# B&R Automation Studio project NAELD004C00R10L518F00 (part 13)

#### Act_OptP0932MagConv3FB.st
```iecst
ACTION Act_OptP0932MagConv3FB:

	//Magazine Conveyor
	IF tyP0932MagConv3.tyFB.tyBtnStop.bRtCompl = TRUE THEN
		eMagConv2Clp3Act	:= MagConv2ClpActStop;

		IF p_eMagConv2Clp3Stat = MagConv2ClpActStop AND p_eMagConv2Clp3Status = Done THEN
			eMagConv2Clp3Act	:= MagConv2ClpActIdle;

			tyP0932MagConv3.tyFB.tyBtnEnt.bRtCompl	:= FALSE;
			tyP0932MagConv3.tyFB.tyBtnEnt.bValue	:= FALSE;
			tyP0932MagConv3.tyFB.tyBtnEnt.bRtLk		:= FALSE;

			tyP0932MagConv3.tyFB.tyBtnExit.bRtCompl	:= FALSE;
			tyP0932MagConv3.tyFB.tyBtnExit.bValue	:= FALSE;
			tyP0932MagConv3.tyFB.tyBtnExit.bRtLk	:= FALSE;

			tyP0932MagConv3.tyFB.tyBtnStop.bRtCompl	:= FALSE;
			tyP0932MagConv3.tyFB.tyBtnStop.bValue	:= TRUE;
			tyP0932MagConv3.tyFB.tyBtnStop.bRtLk	:= TRUE;
		END_IF

	ELSIF tyP0932MagConv3.tyFB.tyBtnEnt.bRtCompl = TRUE THEN
		tyP0932MagConv3.tyFB.tyBtnEnt.bValue	:= TRUE;
		tyP0932MagConv3.tyFB.tyBtnEnt.bRtLk		:= TRUE;

		tyP0932MagConv3.tyFB.tyBtnStop.bValue	:= FALSE;
		tyP0932MagConv3.tyFB.tyBtnStop.bRtLk	:= FALSE;

		eMagConv2Clp3Act	:= MagConv2ClpActEnt;

		IF p_eMagConv2Clp3Stat = MagConv2ClpActEnt AND p_eMagConv2Clp3Status = Done THEN
			eMagConv2Clp3Act	:= MagConv2ClpActIdle;

			tyP0932MagConv3.tyFB.tyBtnEnt.bRtCompl	:= FALSE;

			tyP0932MagConv3.tyFB.tyBtnEnt.bValue	:= FALSE;
			tyP0932MagConv3.tyFB.tyBtnEnt.bRtLk		:= FALSE;

			tyP0932MagConv3.tyFB.tyBtnStop.bValue	:= TRUE;
			tyP0932MagConv3.tyFB.tyBtnStop.bRtLk	:= TRUE;
		END_IF

	ELSIF (p_eMagConv2Clp3Stat = MagConv2ClpActPreExit AND p_eMagConv2Clp3Status = Done) THEN
		eMagConv2Clp3Act	:= MagConv2ClpActIdle;

		tyP0932MagConv3.tyFB.tyBtnExit.bRtCompl	:= FALSE;

		tyP0932MagConv3.tyFB.tyBtnExit.bValue	:= FALSE;
		tyP0932MagConv3.tyFB.tyBtnExit.bRtLk	:= FALSE;

		tyP0932MagConv3.tyFB.tyBtnStop.bValue	:= TRUE;
		tyP0932MagConv3.tyFB.tyBtnStop.bRtLk	:= TRUE;

	ELSIF (p_eMagConv2Clp3Stat = MagConv2ClpActExit AND p_eMagConv2Clp3Status = Done) THEN
		eMagConv2Clp3Act	:= MagConv2ClpActIdle;

		tyP0932MagConv3.tyFB.tyBtnExit.bRtCompl	:= FALSE;

		tyP0932MagConv3.tyFB.tyBtnExit.bValue	:= FALSE;
		tyP0932MagConv3.tyFB.tyBtnExit.bRtLk	:= FALSE;

		tyP0932MagConv3.tyFB.tyBtnStop.bValue	:= TRUE;
		tyP0932MagConv3.tyFB.tyBtnStop.bRtLk	:= TRUE;

	ELSIF tyP0932MagConv3.tyFB.tyBtnExit.bRtCompl = TRUE THEN
		tyP0932MagConv3.tyFB.tyBtnExit.bRtCompl	:= FALSE;
		tyP0932MagConv3.tyFB.tyBtnExit.bValue	:= TRUE;
		tyP0932MagConv3.tyFB.tyBtnExit.bRtLk	:= TRUE;

		tyP0932MagConv3.tyFB.tyBtnStop.bValue	:= FALSE;
		tyP0932MagConv3.tyFB.tyBtnStop.bRtLk	:= FALSE;

		IF p_tyDI.bMagConvEntSen3  THEN
			eMagConv2Clp3Act	:= MagConv2ClpActExit;
		ELSE
			IF p_tyDI.bMagPresentSen3 THEN
				eMagConv2Clp3Act	:= MagConv2ClpActPreExit;
			ELSE
				eMagConv2Clp3Act	:= MagConv2ClpActExit;
			END_IF
		END_IF
	END_IF

	//Magazine Clamper
	IF tyP0932MagConv3.tyCom.tyBtnSwitch.bValue = FALSE THEN

		//Fixed/Bottom
		IF tyP0932MagConv3.tyFB.tyBtnFixedUnclamp.bRtCompl = TRUE THEN
			tyP0932MagConv3.tyFB.tyBtnFixedUnclamp.bRtCompl	:= FALSE;

			tyP0932MagConv3.tyFB.tyBtnFixedUnclamp.bValue	:= TRUE;
			tyP0932MagConv3.tyFB.tyBtnFixedClamp.bValue		:= FALSE;

		ELSIF tyP0932MagConv3.tyFB.tyBtnFixedClamp.bRtCompl = TRUE THEN
			tyP0932MagConv3.tyFB.tyBtnFixedClamp.bRtCompl	:= FALSE;

			tyP0932MagConv3.tyFB.tyBtnFixedClamp.bValue		:= TRUE;
			tyP0932MagConv3.tyFB.tyBtnFixedUnclamp.bValue	:= FALSE;

		END_IF

		//Remote/Top
		IF tyP0932MagConv3.tyFB.tyBtnRemoteUnclamp.bRtCompl = TRUE THEN
			tyP0932MagConv3.tyFB.tyBtnRemoteUnclamp.bRtCompl	:= FALSE;

			tyP0932MagConv3.tyFB.tyBtnRemoteUnclamp.bValue	:= TRUE;
			tyP0932MagConv3.tyFB.tyBtnRemoteClamp.bValue	:= FALSE;

		ELSIF tyP0932MagConv3.tyFB.tyBtnRemoteClamp.bRtCompl = TRUE THEN
			tyP0932MagConv3.tyFB.tyBtnRemoteClamp.bRtCompl	:= FALSE;

			tyP0932MagConv3.tyFB.tyBtnRemoteClamp.bValue	:= TRUE;
			tyP0932MagConv3.tyFB.tyBtnRemoteUnclamp.bValue	:= FALSE;

		END_IF

		//Selection
		IF tyP0932MagConv3.tyFB.tyBtnSelUnclamp.bRtCompl = TRUE THEN
			tyP0932MagConv3.tyFB.tyBtnSelUnclamp.bRtCompl	:= FALSE;

			tyP0932MagConv3.tyFB.tyBtnSelUnclamp.bValue	:= TRUE;
			tyP0932MagConv3.tyFB.tyBtnSelClamp.bValue	:= FALSE;

		ELSIF tyP0932MagConv3.tyFB.tyBtnSelClamp.bRtCompl = TRUE THEN
			tyP0932MagConv3.tyFB.tyBtnSelClamp.bRtCompl	:= FALSE;

			tyP0932MagConv3.tyFB.tyBtnSelClamp.bValue	:= TRUE;
			tyP0932MagConv3.tyFB.tyBtnSelUnclamp.bValue	:= FALSE;

		END_IF

		// Fixed Clamper
		IF tyP0932MagConv3.tyFB.tyBtnFixedUnclamp.bValue = TRUE THEN

			eMagConv2Clp3Act	:= MagConv2ClpActFixClprUnclamp;

			IF p_eMagConv2Clp3Stat = MagConv2ClpActFixClprUnclamp AND p_eMagConv2Clp3Status = Done THEN

				eMagConv2Clp3Act	:= MagConv2ClpActIdle;

				tyP0932MagConv3.tyFB.tyBtnFixedUnclamp.bValue	:= FALSE;

			ELSIF p_eMagConv2Clp3Status = Error THEN

				tyP0932MagConv3.tyFB.tyBtnFixedUnclamp.bValue	:= FALSE;

			END_IF

		ELSIF tyP0932MagConv3.tyFB.tyBtnFixedClamp.bValue = TRUE THEN
			eMagConv2Clp3Act	:= MagConv2ClpActFixClprClamp;

			IF p_eMagConv2Clp3Stat = MagConv2ClpActFixClprClamp AND p_eMagConv2Clp3Status = Done THEN

				eMagConv2Clp3Act	:= MagConv2ClpActIdle;

				tyP0932MagConv3.tyFB.tyBtnFixedClamp.bValue := FALSE;

			ELSIF p_eMagConv2Clp3Status = Error THEN

				tyP0932MagConv3.tyFB.tyBtnFixedClamp.bValue := FALSE;

			END_IF

		END_IF

		//Remote Clamper
		IF tyP0932MagConv3.tyFB.tyBtnRemoteUnclamp.bValue = TRUE THEN

			eMagConv2Clp3Act	:= MagConv2ClpActRmtClprUnclamp;

			IF p_eMagConv2Clp3Stat = MagConv2ClpActRmtClprUnclamp AND p_eMagConv2Clp3Status = Done THEN

				eMagConv2Clp3Act	:= MagConv2ClpActIdle;

				tyP0932MagConv3.tyFB.tyBtnRemoteUnclamp.bValue	:= FALSE;

			ELSIF p_eMagConv2Clp3Status = Error THEN

				tyP0932MagConv3.tyFB.tyBtnRemoteUnclamp.bValue	:= FALSE;

			END_IF

		ELSIF tyP0932MagConv3.tyFB.tyBtnRemoteClamp.bValue = TRUE THEN
			eMagConv2Clp3Act	:= MagConv2ClpActRmtClprClamp;

			IF p_eMagConv2Clp3Stat = MagConv2ClpActRmtClprClamp AND p_eMagConv2Clp3Status = Done THEN

				eMagConv2Clp3Act	:= MagConv2ClpActIdle;

				tyP0932MagConv3.tyFB.tyBtnRemoteClamp.bValue := FALSE;

			ELSIF p_eMagConv2Clp3Status = Error THEN
				tyP0932MagConv3.tyFB.tyBtnRemoteClamp.bValue := FALSE;

			END_IF

		END_IF

		//Selection Clamper
		IF tyP0932MagConv3.tyFB.tyBtnSelUnclamp.bValue = TRUE THEN

			eMagConvSelClp3Act	:= PneuActExt;

			IF p_eSelClamp3Stat = PneuActExt AND p_eSelClamp3Status = Done THEN

				eMagConvSelClp3Act	:= PneuActIdle;

				tyP0932MagConv3.tyFB.tyBtnSelUnclamp.bValue	:= FALSE;

			ELSIF p_eSelClamp3Status = Error THEN
				eMagConvSelClp3Act	:= PneuActIdle;
				tyP0932MagConv3.tyFB.tyBtnSelUnclamp.bValue	:= FALSE;

			END_IF

		ELSIF tyP0932MagConv3.tyFB.tyBtnSelClamp.bValue = TRUE THEN
			eMagConvSelClp3Act	:= PneuActRet;

			IF p_eSelClamp3Stat = PneuActRet AND p_eSelClamp3Status = Done THEN

				eMagConvSelClp3Act	:= PneuActIdle;

				tyP0932MagConv3.tyFB.tyBtnSelClamp.bValue	:= FALSE;

			ELSIF p_eSelClamp3Status = Error THEN
				eMagConvSelClp3Act	:= PneuActIdle;
				tyP0932MagConv3.tyFB.tyBtnSelClamp.bValue	:= FALSE;

			END_IF

		END_IF

		//Update Status
		tyP0932MagConv3.tyDC.tyBtnFixedUnclamp.bValue	:= NOT p_bMagConv2Clp3ClprFixClampCtrl;
		tyP0932MagConv3.tyDC.tyBtnFixedClamp.bValue		:= p_bMagConv2Clp3ClprFixClampCtrl;
		tyP0932MagConv3.tyDC.tyBtnRemoteUnclamp.bValue	:= NOT p_bMagConv2Clp3ClprRmtClampCtrl;
		tyP0932MagConv3.tyDC.tyBtnRemoteClamp.bValue	:= p_bMagConv2Clp3ClprRmtClampCtrl;

		tyP0932MagConv3.tyDC.tyBtnSelUnclamp.bRtCompl	:= FALSE;
		tyP0932MagConv3.tyDC.tyBtnSelClamp.bRtCompl		:= FALSE;
		tyP0932MagConv3.tyDC.tyBtnSelUnclamp.bValue	:= p_bSelClamp3RetCtrl;
		tyP0932MagConv3.tyDC.tyBtnSelClamp.bValue	:= p_bSelClamp3ExtCtrl;
	END_IF

	//Mask
	IF p_tyUsrMgmtCurrAccessRgt.bManualFBOnly THEN

		fUIInRtStatOff(ADR(tyP0932MagConv3.tyCom.tyBtnSwitch.uiMaskRtStat));

	ELSE

		IF p_eMagConv2Clp3Status = Error THEN

			fUIInRtStatOff(ADR(tyP0932MagConv3.tyFB.tyBtnEnt.uiMaskRtStat));
			fUIInRtStatOff(ADR(tyP0932MagConv3.tyFB.tyBtnExit.uiMaskRtStat));
			fUIInRtStatOff(ADR(tyP0932MagConv3.tyFB.tyBtnFixedClamp.uiMaskRtStat));
			fUIInRtStatOff(ADR(tyP0932MagConv3.tyFB.tyBtnFixedUnclamp.uiMaskRtStat));
			fUIInRtStatOff(ADR(tyP0932MagConv3.tyFB.tyBtnRemoteClamp.uiMaskRtStat));
			fUIInRtStatOff(ADR(tyP0932MagConv3.tyFB.tyBtnRemoteUnclamp.uiMaskRtStat));
			fUIInRtStatOff(ADR(tyP0932MagConv3.tyFB.tyBtnSelClamp.uiMaskRtStat));
			fUIInRtStatOff(ADR(tyP0932MagConv3.tyFB.tyBtnSelUnclamp.uiMaskRtStat));
			fUIInRtStatHide(ADR(tyP0932MagConv3.tyCom.tyBtnSwitch.uiMaskRtStat));

		ELSIF tyP0932MagConv3.tyFB.tyBtnEnt.bRtCompl = TRUE THEN

			fUIInRtStatHide(ADR(tyP0932MagConv3.tyFB.tyBtnEnt.uiMaskRtStat));
			fUIInRtStatOff(ADR(tyP0932MagConv3.tyFB.tyBtnExit.uiMaskRtStat));
			fUIInRtStatOff(ADR(tyP0932MagConv3.tyFB.tyBtnFixedClamp.uiMaskRtStat));
			fUIInRtStatOff(ADR(tyP0932MagConv3.tyFB.tyBtnFixedUnclamp.uiMaskRtStat));
			fUIInRtStatOff(ADR(tyP0932MagConv3.tyFB.tyBtnRemoteClamp.uiMaskRtStat));
			fUIInRtStatOff(ADR(tyP0932MagConv3.tyFB.tyBtnRemoteUnclamp.uiMaskRtStat));
			fUIInRtStatOff(ADR(tyP0932MagConv3.tyFB.tyBtnSelClamp.uiMaskRtStat));
			fUIInRtStatOff(ADR(tyP0932MagConv3.tyFB.tyBtnSelUnclamp.uiMaskRtStat));
			fUIInRtStatOff(ADR(tyP0932MagConv3.tyCom.tyBtnSwitch.uiMaskRtStat));

		ELSIF tyP0932MagConv3.tyFB.tyBtnExit.bRtCompl = TRUE THEN

			fUIInRtStatOff(ADR(tyP0932MagConv3.tyFB.tyBtnEnt.uiMaskRtStat));
			fUIInRtStatHide(ADR(tyP0932MagConv3.tyFB.tyBtnExit.uiMaskRtStat));
			fUIInRtStatOff(ADR(tyP0932MagConv3.tyFB.tyBtnFixedClamp.uiMaskRtStat));
			fUIInRtStatOff(ADR(tyP0932MagConv3.tyFB.tyBtnFixedUnclamp.uiMaskRtStat));
			fUIInRtStatOff(ADR(tyP0932MagConv3.tyFB.tyBtnRemoteClamp.uiMaskRtStat));
			fUIInRtStatOff(ADR(tyP0932MagConv3.tyFB.tyBtnRemoteUnclamp.uiMaskRtStat));
			fUIInRtStatOff(ADR(tyP0932MagConv3.tyFB.tyBtnSelClamp.uiMaskRtStat));
			fUIInRtStatOff(ADR(tyP0932MagConv3.tyFB.tyBtnSelUnclamp.uiMaskRtStat));
			fUIInRtStatOff(ADR(tyP0932MagConv3.tyCom.tyBtnSwitch.uiMaskRtStat));

		ELSIF tyP0932MagConv3.tyFB.tyBtnFixedClamp.bValue = TRUE OR tyP0932MagConv3.tyFB.tyBtnRemoteClamp.bValue = TRUE
			OR tyP0932MagConv3.tyFB.tyBtnFixedUnclamp.bValue = TRUE OR tyP0932MagConv3.tyFB.tyBtnRemoteUnclamp.bValue = TRUE
			OR tyP0932MagConv3.tyFB.tyBtnSelClamp.bValue = TRUE OR tyP0932MagConv3.tyFB.tyBtnSelUnclamp.bValue = TRUE
			THEN

			fUIInRtStatOff(ADR(tyP0932MagConv3.tyFB.tyBtnEnt.uiMaskRtStat));
			fUIInRtStatOff(ADR(tyP0932MagConv3.tyFB.tyBtnExit.uiMaskRtStat));
			fUIInRtStatHide(ADR(tyP0932MagConv3.tyFB.tyBtnFixedClamp.uiMaskRtStat));
			fUIInRtStatHide(ADR(tyP0932MagConv3.tyFB.tyBtnFixedUnclamp.uiMaskRtStat));
			fUIInRtStatHide(ADR(tyP0932MagConv3.tyFB.tyBtnRemoteClamp.uiMaskRtStat));
			fUIInRtStatHide(ADR(tyP0932MagConv3.tyFB.tyBtnRemoteUnclamp.uiMaskRtStat));
			fUIInRtStatHide(ADR(tyP0932MagConv3.tyFB.tyBtnSelClamp.uiMaskRtStat));
			fUIInRtStatHide(ADR(tyP0932MagConv3.tyFB.tyBtnSelUnclamp.uiMaskRtStat));
			fUIInRtStatOff(ADR(tyP0932MagConv3.tyCom.tyBtnSwitch.uiMaskRtStat));

		ELSE

			fUIInRtStatHide(ADR(tyP0932MagConv3.tyFB.tyBtnEnt.uiMaskRtStat));
			fUIInRtStatHide(ADR(tyP0932MagConv3.tyFB.tyBtnExit.uiMaskRtStat));
			fUIInRtStatHide(ADR(tyP0932MagConv3.tyFB.tyBtnFixedClamp.uiMaskRtStat));
			fUIInRtStatHide(ADR(tyP0932MagConv3.tyFB.tyBtnFixedUnclamp.uiMaskRtStat));
			fUIInRtStatHide(ADR(tyP0932MagConv3.tyFB.tyBtnRemoteClamp.uiMaskRtStat));
			fUIInRtStatHide(ADR(tyP0932MagConv3.tyFB.tyBtnRemoteUnclamp.uiMaskRtStat));
			fUIInRtStatHide(ADR(tyP0932MagConv3.tyFB.tyBtnSelClamp.uiMaskRtStat));
			fUIInRtStatHide(ADR(tyP0932MagConv3.tyFB.tyBtnSelUnclamp.uiMaskRtStat));
			fUIInRtStatHide(ADR(tyP0932MagConv3.tyCom.tyBtnSwitch.uiMaskRtStat));

		END_IF
	END_IF

	IF p_tyDI.bMagConvCAB717MagSen3 THEN
		fUIInRtStatOff(ADR(tyP0932MagConv3.tyFB.tyBtnSelClamp.uiMaskRtStat));
	END_IF

END_ACTION
```

#### Act_OptP0932MagConv3FBStat.st
```iecst
ACTION Act_OptP0932MagConv3FBStat:

	IF tyP0932MagConv3.tyFB.tyBtnFixedClamp.bValue = TRUE OR tyP0932MagConv3.tyFB.tyBtnRemoteClamp.bValue = TRUE
		OR tyP0932MagConv3.tyFB.tyBtnFixedUnclamp.bValue = TRUE OR tyP0932MagConv3.tyFB.tyBtnRemoteUnclamp.bValue = TRUE
		THEN
		tyP0932MagConv3.tyFB.tyStringStat.sValue	:= p_sMagConv2Clp3StatTxt;
	ELSIF tyP0932MagConv3.tyFB.tyBtnSelUnclamp.bValue = TRUE OR tyP0932MagConv3.tyFB.tyBtnSelClamp.bValue = TRUE
		THEN
		tyP0932MagConv3.tyFB.tyStringStat.sValue	:= p_sSelClamp3StatTxt;
	END_IF
END_ACTION
```

#### Act_OptP0932MagConv3Sen.st
```iecst
ACTION Act_OptP0932MagConv3Sen:

	tyP0932MagConv3.tyCom.tyBtnMagPresentSen.bValue			:= p_tyDI.bMagPresentSen3;
	tyP0932MagConv3.tyCom.tyBtnMagConvEntSen.bValue			:= p_tyDI.bMagConvEntSen3;
	tyP0932MagConv3.tyCom.tyBtnMagAIVPosSen1.bValue			:= p_tyDI.bMag3AGVInPosSen1;
	tyP0932MagConv3.tyCom.tyBtnMagAIVPosSen2.bValue			:= p_tyDI.bMag3AGVInPosSen2;
	tyP0932MagConv3.tyCom.tyBtnMagOrientationChkSen1.bValue	:= p_tyDI.bMag3OrientChkSen1;
	tyP0932MagConv3.tyCom.tyBtnMagOrientationChkSen2.bValue	:= p_tyDI.bMag3OrientChkSen2;

	tyP0932MagConv3.tyCom.tyBtnFixedClampRS.bValue			:= p_tyDI.bMag3FixedClampRS;
	tyP0932MagConv3.tyCom.tyBtnFixedUnclampRS.bValue		:= p_tyDI.bMag3FixedUnclampRS;
	tyP0932MagConv3.tyCom.tyBtnRemoteClampRS.bValue			:= p_tyDI.bMag3RemoteClampRS;
	tyP0932MagConv3.tyCom.tyBtnRemoteUnclampRS.bValue		:= p_tyDI.bMag3RemoteUnclampRS;

	tyP0932MagConv3.tyCom.tyBtnSelUnclampRS.bValue			:= p_tyDI.bMag3SelUnClampRS;

	tyP0932MagConv3.tyCom.tyBtnCAB717Sen.bValue				:= p_tyDI.bMagConvCAB717MagSen3;
	tyP0932MagConv3.tyCom.tyBtnHeightSen.bValue				:= p_tyDI.bMagConvHeightSen3 OR p_tyDI.bHighMagDetSen3;
	tyP0932MagConv3.tyCom.tyBtnMagSmallSen.bValue			:= p_tyDI.bMagConvSmallMagSen3;
	tyP0932MagConv3.tyCom.tyBtnMagLargeSen.bValue			:= p_tyDI.bMagConvLargeMagSen3;
	tyP0932MagConv3.tyCom.tyBtnMagDetSen.bValue				:= p_tyDI.bMag3FixedSideDetect;

	//Machine Bitmap //23
//	IF p_tyNtParamCurr.bMagAutoVerifyPrep = FALSE THEN
//		IF tyP0932MagConv3.tyFB.tyBtnFixedClamp.bRtCompl OR  tyP0932MagConv3.tyFB.tyBtnRemoteClamp.bRtCompl
//			OR tyP0932MagConv3.tyDC.tyBtnFixedClamp.bRtCompl OR tyP0932MagConv3.tyDC.tyBtnRemoteClamp.bRtCompl  THEN
//
//			tyP0932MagConv3.tyCom.tyBitmapMc.uiValueIdx	:= 2;
//
//		ELSIF tyP0932MagConv3.tyFB.tyBtnFixedUnclamp.bRtCompl OR tyP0932MagConv3.tyFB.tyBtnRemoteUnclamp.bRtCompl
//			OR tyP0932MagConv3.tyDC.tyBtnFixedUnclamp.bRtCompl OR tyP0932MagConv3.tyDC.tyBtnRemoteUnclamp.bRtCompl  THEN
//
//			tyP0932MagConv3.tyCom.tyBitmapMc.uiValueIdx	:= 1;
//
//		ELSIF tyP0932MagConv3.tyFB.tyBtnEnt.bRtCompl OR tyP0932MagConv3.tyFB.tyBtnExit.bRtCompl OR tyP0932MagConv3.tyFB.tyBtnStop.bRtCompl
//			OR tyP0932MagConv3.tyDC.tyBtnMagIn.bRtCompl OR tyP0932MagConv3.tyDC.tyBtnMagOut.bRtCompl OR tyP0932MagConv3.tyDC.tyBtnStop.bRtCompl THEN
//
//			tyP0932MagConv3.tyCom.tyBitmapMc.uiValueIdx	:= 0;
//
//		END_IF

	IF p_tyNtParamCurr.eProjMag = LDMagTriple AND p_tyNtParamCurr.bProjCurtainSenPrep = FALSE AND p_tyNtParamCurr.eCustomerReq <> Siemens AND p_tyNtParamCurr.eCustomerReq <> We_Fabricate  THEN
		IF tyP0932MagConv3.tyFB.tyBtnFixedClamp.bRtCompl
			OR tyP0932MagConv3.tyDC.tyBtnFixedClamp.bRtCompl THEN

			tyP0932MagConv3.tyCom.tyBitmapMc.uiValueIdx	:= 2;

		ELSIF tyP0932MagConv3.tyFB.tyBtnFixedUnclamp.bRtCompl
			OR tyP0932MagConv3.tyDC.tyBtnFixedUnclamp.bRtCompl THEN

			tyP0932MagConv3.tyCom.tyBitmapMc.uiValueIdx	:= 1;

		ELSIF tyP0932MagConv3.tyFB.tyBtnRemoteClamp.bRtCompl
			OR tyP0932MagConv3.tyDC.tyBtnRemoteClamp.bRtCompl THEN

			tyP0932MagConv3.tyCom.tyBitmapMc.uiValueIdx	:= 14;

		ELSIF tyP0932MagConv3.tyFB.tyBtnRemoteUnclamp.bRtCompl
			OR tyP0932MagConv3.tyDC.tyBtnRemoteUnclamp.bRtCompl THEN

			tyP0932MagConv3.tyCom.tyBitmapMc.uiValueIdx	:= 13;

		ELSIF tyP0932MagConv3.tyFB.tyBtnSelClamp.bRtCompl
			OR tyP0932MagConv3.tyDC.tyBtnSelClamp.bRtCompl THEN

			tyP0932MagConv3.tyCom.tyBitmapMc.uiValueIdx	:= 20;

		ELSIF tyP0932MagConv3.tyFB.tyBtnSelUnclamp.bRtCompl
			OR tyP0932MagConv3.tyDC.tyBtnSelUnclamp.bRtCompl THEN

			tyP0932MagConv3.tyCom.tyBitmapMc.uiValueIdx	:= 19;

		ELSIF tyP0932MagConv3.tyFB.tyBtnEnt.bRtCompl OR tyP0932MagConv3.tyFB.tyBtnExit.bRtCompl OR tyP0932MagConv3.tyFB.tyBtnStop.bRtCompl
			OR tyP0932MagConv3.tyDC.tyBtnMagIn.bRtCompl OR tyP0932MagConv3.tyDC.tyBtnMagOut.bRtCompl OR tyP0932MagConv3.tyDC.tyBtnStop.bRtCompl THEN

			tyP0932MagConv3.tyCom.tyBitmapMc.uiValueIdx	:= 0;

		END_IF
	ELSIF p_tyNtParamCurr.eProjMag = LDMagTriple AND p_tyNtParamCurr.bProjCurtainSenPrep OR p_tyNtParamCurr.eCustomerReq = Siemens OR p_tyNtParamCurr.eCustomerReq = We_Fabricate THEN
		tyP0932MagConv3.tyCom.tyBitmapMc.uiValueIdx	:= 386-23;

	ELSIF p_tyNtParamCurr.eProjMag = LDMagQuadruple AND p_tyNtParamCurr.bMagAutoVerifyPrep THEN
		IF tyP0932MagConv3.tyFB.tyBtnFixedClamp.bRtCompl
			OR tyP0932MagConv3.tyDC.tyBtnFixedClamp.bRtCompl THEN

			tyP0932MagConv3.tyCom.tyBitmapMc.uiValueIdx	:= 111;

		ELSIF tyP0932MagConv3.tyFB.tyBtnFixedUnclamp.bRtCompl
			OR tyP0932MagConv3.tyDC.tyBtnFixedUnclamp.bRtCompl THEN

			tyP0932MagConv3.tyCom.tyBitmapMc.uiValueIdx	:= 110;

		ELSIF tyP0932MagConv3.tyFB.tyBtnRemoteClamp.bRtCompl
			OR tyP0932MagConv3.tyDC.tyBtnRemoteClamp.bRtCompl THEN

			tyP0932MagConv3.tyCom.tyBitmapMc.uiValueIdx	:= 113;

		ELSIF tyP0932MagConv3.tyFB.tyBtnRemoteUnclamp.bRtCompl
			OR tyP0932MagConv3.tyDC.tyBtnRemoteUnclamp.bRtCompl THEN

			tyP0932MagConv3.tyCom.tyBitmapMc.uiValueIdx	:= 112;

		ELSIF tyP0932MagConv3.tyFB.tyBtnSelClamp.bRtCompl
			OR tyP0932MagConv3.tyDC.tyBtnSelClamp.bRtCompl THEN

			tyP0932MagConv3.tyCom.tyBitmapMc.uiValueIdx	:= 115;

		ELSIF tyP0932MagConv3.tyFB.tyBtnSelUnclamp.bRtCompl
			OR tyP0932MagConv3.tyDC.tyBtnSelUnclamp.bRtCompl THEN

			tyP0932MagConv3.tyCom.tyBitmapMc.uiValueIdx	:= 114;

		ELSIF tyP0932MagConv3.tyFB.tyBtnEnt.bRtCompl OR tyP0932MagConv3.tyFB.tyBtnExit.bRtCompl OR tyP0932MagConv3.tyFB.tyBtnStop.bRtCompl
			OR tyP0932MagConv3.tyDC.tyBtnMagIn.bRtCompl OR tyP0932MagConv3.tyDC.tyBtnMagOut.bRtCompl OR tyP0932MagConv3.tyDC.tyBtnStop.bRtCompl THEN

			tyP0932MagConv3.tyCom.tyBitmapMc.uiValueIdx	:= 109;

		END_IF
	END_IF

	IF p_tyNtParamCurr.eProjMag = LDMagTriple AND p_tyNtParamCurr.bMagAutoVerifyPrep = FALSE AND p_tyNtParamCurr.bProjMotorizedPullerPrep = FALSE THEN
		IF tyP0932MagConv3.tyCom.tyBitmapMc.uiValueIdx < 100 THEN
			tyP0932MagConv3.tyCom.tyBitmapMc.uiValueIdx	:= tyP0932MagConv3.tyCom.tyBitmapMc.uiValueIdx + 100;
		END_IF
	ELSIF p_tyNtParamCurr.eProjMag = LDMagDual AND p_tyNtParamCurr.bMagAutoVerifyPrep = TRUE THEN
		IF tyP0932MagConv3.tyCom.tyBitmapMc.uiValueIdx < 200 THEN
			tyP0932MagConv3.tyCom.tyBitmapMc.uiValueIdx	:= tyP0932MagConv3.tyCom.tyBitmapMc.uiValueIdx + 200;
		END_IF
	ELSIF p_tyNtParamCurr.eProjMag = LDMagTriple AND p_tyNtParamCurr.bMagAutoVerifyPrep = FALSE AND p_tyNtParamCurr.bProjMotorizedPullerPrep = TRUE THEN
			IF tyP0932MagConv3.tyCom.tyBitmapMc.uiValueIdx < 300 THEN
				tyP0932MagConv3.tyCom.tyBitmapMc.uiValueIdx	:= tyP0932MagConv3.tyCom.tyBitmapMc.uiValueIdx + 300;
			END_IF
	END_IF

END_ACTION
```

#### Act_OptP0932Navi.st
```iecst
ACTION Act_OptP0932Navi:

	CASE p_tyNtParamCurr.eProjMag OF
		LDMagDual:
			IF tyP0932MagConv3.tyNavi3Lyr3.tyBtnBack.bRtCompl = TRUE THEN
				tyP0932MagConv3.tyNavi3Lyr3.tyBtnBack.bRtCompl	:= FALSE;
				tyP0932MagConv3.tyNavi3Lyr3.tyBtnBack.bValue	:= FALSE;

				eChgPage	:= UIP0920MtrNPneuCtrl;

				bDispMagConv1	:= FALSE;
				bDispMagConv2	:= FALSE;
				bDispMagConv3	:= TRUE;
				bDispMagConv4	:= FALSE;

			ELSIF tyP0932MagConv3.tyNavi3Lyr3.tyBtnLeft.bRtCompl = TRUE
				OR tyP0932MagConv3.tyNavi3Lyr3.tyBtnRgt.bRtCompl = TRUE
				THEN
				tyP0932MagConv3.tyNavi3Lyr3.tyBtnLeft.bRtCompl			:= FALSE;
				tyP0932MagConv3.tyNavi3Lyr3.tyBtnLeft.bValue			:= FALSE;
				tyP0932MagConv3.tyNavi3Lyr3.tyBtnRgt.bRtCompl			:= FALSE;
				tyP0932MagConv3.tyNavi3Lyr3.tyBtnRgt.bValue				:= FALSE;
				eChgPage												:= UIP0931MagConv2;
				bDispMagConv1	:= FALSE;
				bDispMagConv2	:= TRUE;
				bDispMagConv3	:= FALSE;
				bDispMagConv4	:= FALSE;
			END_IF

		LDMagTriple:
			IF tyP0932MagConv3.tyNavi3Lyr3.tyBtnBack.bRtCompl = TRUE THEN
				tyP0932MagConv3.tyNavi3Lyr3.tyBtnBack.bRtCompl	:= FALSE;
				tyP0932MagConv3.tyNavi3Lyr3.tyBtnBack.bValue	:= FALSE;

				eChgPage	:= UIP0920MtrNPneuCtrl;

				bDispMagConv1	:= FALSE;
				bDispMagConv2	:= FALSE;
				bDispMagConv3	:= TRUE;
				bDispMagConv4	:= FALSE;

			ELSIF tyP0932MagConv3.tyNavi3Lyr3.tyBtnLeft.bRtCompl = TRUE THEN
				tyP0932MagConv3.tyNavi3Lyr3.tyBtnLeft.bRtCompl			:= FALSE;
				tyP0932MagConv3.tyNavi3Lyr3.tyBtnLeft.bValue			:= FALSE;
				eChgPage												:= UIP0931MagConv2;
				bDispMagConv1	:= FALSE;
				bDispMagConv2	:= TRUE;
				bDispMagConv3	:= FALSE;
				bDispMagConv4	:= FALSE;

			ELSIF tyP0932MagConv3.tyNavi3Lyr3.tyBtnRgt.bRtCompl = TRUE THEN
				tyP0932MagConv3.tyNavi3Lyr3.tyBtnRgt.bRtCompl			:= FALSE;
				tyP0932MagConv3.tyNavi3Lyr3.tyBtnRgt.bValue				:= FALSE;
				eChgPage												:= UIP0930MagConv1;
				bDispMagConv1	:= TRUE;
				bDispMagConv2	:= FALSE;
				bDispMagConv3	:= FALSE;
				bDispMagConv4	:= FALSE;
			END_IF

		LDMagQuadruple:
			IF tyP0932MagConv3.tyNavi4Lyr3.tyBtnBack.bRtCompl = TRUE THEN
				tyP0932MagConv3.tyNavi4Lyr3.tyBtnBack.bRtCompl	:= FALSE;
				tyP0932MagConv3.tyNavi4Lyr3.tyBtnBack.bValue	:= FALSE;

				eChgPage	:= UIP0920MtrNPneuCtrl;
				bDispMagConv1	:= FALSE;
				bDispMagConv2	:= FALSE;
				bDispMagConv3	:= TRUE;
				bDispMagConv4	:= FALSE;

			ELSIF tyP0932MagConv3.tyNavi4Lyr3.tyBtnLeft.bRtCompl = TRUE THEN
				tyP0932MagConv3.tyNavi4Lyr3.tyBtnLeft.bRtCompl			:= FALSE;
				tyP0932MagConv3.tyNavi4Lyr3.tyBtnLeft.bValue			:= FALSE;
				eChgPage												:= UIP0931MagConv2;
				bDispMagConv1	:= FALSE;
				bDispMagConv2	:= TRUE;
				bDispMagConv3	:= FALSE;
				bDispMagConv4	:= FALSE;

			ELSIF tyP0932MagConv3.tyNavi4Lyr3.tyBtnRgt.bRtCompl = TRUE THEN
				tyP0932MagConv3.tyNavi4Lyr3.tyBtnRgt.bRtCompl			:= FALSE;
				tyP0932MagConv3.tyNavi4Lyr3.tyBtnRgt.bValue				:= FALSE;
				eChgPage												:= UIP0939MagConv4;
				bDispMagConv1	:= FALSE;
				bDispMagConv2	:= FALSE;
				bDispMagConv3	:= FALSE;
				bDispMagConv4	:= TRUE;
			END_IF
	END_CASE

END_ACTION
```

#### Act_OptP0932RstMnl.st
```iecst
ACTION Act_OptP0932RstMnl:

	IF EDGEPOS((bManualMod = FALSE) OR (p_eMagConv2Clp3Status = Error)) THEN

		eMagConv2Clp3Act	:= MagConv2ClpActIdle;
		eMagConvSelClp3Act	:= PneuActIdle;
		//Magazine Conveyor
		//FB
		tyP0932MagConv3.tyFB.tyBtnEnt.bRtCompl				:= FALSE;
		tyP0932MagConv3.tyFB.tyBtnExit.bRtCompl				:= FALSE;
		tyP0932MagConv3.tyFB.tyBtnStop.bRtCompl				:= FALSE;

		tyP0932MagConv3.tyFB.tyBtnEnt.bValue				:= FALSE;
		tyP0932MagConv3.tyFB.tyBtnExit.bValue				:= FALSE;
		tyP0932MagConv3.tyFB.tyBtnStop.bValue				:= TRUE;

		tyP0932MagConv3.tyFB.tyBtnEnt.bRtLk					:= FALSE;
		tyP0932MagConv3.tyFB.tyBtnExit.bRtLk				:= FALSE;
		tyP0932MagConv3.tyFB.tyBtnStop.bRtLk				:= TRUE;

		tyP0932MagConv3.tyFB.tyBtnEnt.uiMaskRtStat.0		:= TRUE;
		tyP0932MagConv3.tyFB.tyBtnExit.uiMaskRtStat.0		:= TRUE;
		tyP0932MagConv3.tyCom.tyBtnSwitch.uiMaskRtStat.0	:= TRUE;

		//Direct
		tyP0932MagConv3.tyDC.tyBtnMagIn.bRtCompl			:= FALSE;
		tyP0932MagConv3.tyDC.tyBtnMagOut.bRtCompl			:= FALSE;
		tyP0932MagConv3.tyDC.tyBtnStop.bRtCompl				:= FALSE;

		tyP0932MagConv3.tyDC.tyBtnMagIn.bValue				:= FALSE;
		tyP0932MagConv3.tyDC.tyBtnMagOut.bValue				:= FALSE;
		tyP0932MagConv3.tyDC.tyBtnStop.bValue				:= TRUE;

		tyP0932MagConv3.tyDC.tyBtnMagIn.bRtLk				:= FALSE;
		tyP0932MagConv3.tyDC.tyBtnMagOut.bRtLk				:= FALSE;
		tyP0932MagConv3.tyDC.tyBtnStop.bRtLk				:= TRUE;

		tyP0932MagConv3.tyDC.tyBtnMagIn.uiMaskRtStat.0		:= TRUE;
		tyP0932MagConv3.tyDC.tyBtnMagOut.uiMaskRtStat.0		:= TRUE;
		tyP0932MagConv3.tyCom.tyBtnSwitch.uiMaskRtStat.0	:= TRUE;

		//Magazine Clamper
		//FB
		//Fixed/Bottom
		tyP0932MagConv3.tyFB.tyBtnFixedClamp.bRtCompl			:= FALSE;
		tyP0932MagConv3.tyFB.tyBtnFixedUnclamp.bRtCompl			:= FALSE;

		tyP0932MagConv3.tyFB.tyBtnFixedClamp.bValue				:= FALSE;
		tyP0932MagConv3.tyFB.tyBtnFixedUnclamp.bValue			:= FALSE;

		//Remote/Top
		tyP0932MagConv3.tyFB.tyBtnRemoteClamp.bRtCompl			:= FALSE;
		tyP0932MagConv3.tyFB.tyBtnRemoteUnclamp.bRtCompl		:= FALSE;

		tyP0932MagConv3.tyFB.tyBtnRemoteClamp.bValue			:= FALSE;
		tyP0932MagConv3.tyFB.tyBtnRemoteUnclamp.bValue			:= FALSE;

		//Selection
		tyP0932MagConv3.tyFB.tyBtnSelClamp.bRtCompl			:= FALSE;
		tyP0932MagConv3.tyFB.tyBtnSelUnclamp.bRtCompl		:= FALSE;

		tyP0932MagConv3.tyFB.tyBtnSelClamp.bValue			:= FALSE;
		tyP0932MagConv3.tyFB.tyBtnSelUnclamp.bValue			:= FALSE;

		tyP0932MagConv3.tyFB.tyBtnFixedClamp.uiMaskRtStat.0		:= TRUE;
		tyP0932MagConv3.tyFB.tyBtnFixedUnclamp.uiMaskRtStat.0	:= TRUE;
		tyP0932MagConv3.tyFB.tyBtnRemoteClamp.uiMaskRtStat.0	:= TRUE;
		tyP0932MagConv3.tyFB.tyBtnRemoteUnclamp.uiMaskRtStat.0	:= TRUE;
		tyP0932MagConv3.tyFB.tyBtnSelClamp.uiMaskRtStat.0		:= TRUE;
		tyP0932MagConv3.tyFB.tyBtnSelUnclamp.uiMaskRtStat.0		:= TRUE;

		tyP0932MagConv3.tyCom.tyBtnSwitch.uiMaskRtStat.0		:= TRUE;

		//Direct
		//Fixed/Bottom
		tyP0932MagConv3.tyDC.tyBtnFixedClamp.bRtCompl			:= FALSE;
		tyP0932MagConv3.tyDC.tyBtnFixedUnclamp.bRtCompl			:= FALSE;

		tyP0932MagConv3.tyDC.tyBtnFixedClamp.bValue				:= FALSE;
		tyP0932MagConv3.tyDC.tyBtnFixedUnclamp.bValue			:= FALSE;

		//Remote/Top
		tyP0932MagConv3.tyDC.tyBtnRemoteClamp.bRtCompl			:= FALSE;
		tyP0932MagConv3.tyDC.tyBtnRemoteUnclamp.bRtCompl		:= FALSE;

		tyP0932MagConv3.tyDC.tyBtnRemoteClamp.bValue			:= FALSE;
		tyP0932MagConv3.tyDC.tyBtnRemoteUnclamp.bValue			:= FALSE;

		//Selection
		tyP0932MagConv3.tyDC.tyBtnSelClamp.bRtCompl				:= FALSE;
		tyP0932MagConv3.tyDC.tyBtnSelUnclamp.bRtCompl			:= FALSE;

		tyP0932MagConv3.tyDC.tyBtnSelClamp.bValue				:= FALSE;
		tyP0932MagConv3.tyDC.tyBtnSelUnclamp.bValue				:= FALSE;

		tyP0932MagConv3.tyDC.tyBtnFixedClamp.uiMaskRtStat.0		:= TRUE;
		tyP0932MagConv3.tyDC.tyBtnFixedUnclamp.uiMaskRtStat.0	:= TRUE;
		tyP0932MagConv3.tyDC.tyBtnRemoteClamp.uiMaskRtStat.0	:= TRUE;
		tyP0932MagConv3.tyDC.tyBtnRemoteUnclamp.uiMaskRtStat.0	:= TRUE;
		tyP0932MagConv3.tyDC.tyBtnSelClamp.uiMaskRtStat.0		:= TRUE;
		tyP0932MagConv3.tyDC.tyBtnSelUnclamp.uiMaskRtStat.0		:= TRUE;

		tyP0932MagConv3.tyCom.tyBtnSwitch.uiMaskRtStat.0		:= TRUE;

	END_IF

	IF EDGEPOS(bManualMod = FALSE) THEN
		tyP0932MagConv3.tyCom.tyBtnSwitch.bValue := FALSE;

		IF p_tyNtParamCurr.bMagAutoVerifyPrep = FALSE THEN
			fUIInRtStatHide(ADR(tyP0932MagConv3.tyDC.tyLyrWithoutSelClamp.uiRtStat));
			fUIInRtStatOff(ADR(tyP0932MagConv3.tyFB.tyLyrWithoutSelClamp.uiRtStat));
		ELSE

			fUIInRtStatHide(ADR(tyP0932MagConv3.tyDC.tyLyr.uiRtStat));
			fUIInRtStatOff(ADR(tyP0932MagConv3.tyFB.tyLyr.uiRtStat));
		END_IF

	END_IF

END_ACTION
```

#### Act_EntP0933Disp.st
```iecst
ACTION Act_EntP0933Disp:

	//Access Address
	p_tyC0002FullMask ACCESS ADR(tyP0933PullConv.tyFullMaskHide);

	p_tyC0004Navi ACCESS ADR(tyP0933PullConv.tyNaviBack);

	p_tyC0005Main ACCESS ADR(tyCommon.tyMain);

	p_tyC0007Notif ACCESS ADR(tyCommon.tyNotif);

	p_tyC0008MsgBox ACCESS ADR(tyP0933PullConv.tyMsgBoxHide);

	p_tyC0009Info ACCESS ADR(tyCommon.tyInfo);

	p_tyP0933PullConvCom ACCESS ADR(tyP0933PullConv.tyCom);
	p_tyP0933PullConvDC ACCESS ADR(tyP0933PullConv.tyDC);
	p_tyP0933PullConvFB ACCESS ADR(tyP0933PullConv.tyFB);

	//Display
	IF p_tyProdRcpCurrRcp0.diMtrPshrExtSpd <> 0 THEN
		tyP0933PullConv.tyFB.tyNumExtSpd.diValue			:= p_tyProdRcpCurrRcp0.diMtrPshrExtSpd;
	ELSE
		tyP0933PullConv.tyFB.tyNumExtSpd.diValue			:= p_tyNtParamCurr.tyProdRcpMtrPshrExtSpd.diMax/2;
	END_IF

	IF p_tyProdRcpCurrRcp0.diMtrPshrExtTorq <> 0 THEN
		tyP0933PullConv.tyFB.tyNumExtTorqPercent.diValue	:= p_tyProdRcpCurrRcp0.diMtrPshrExtTorq;
	ELSE
		tyP0933PullConv.tyFB.tyNumExtTorqPercent.diValue	:= p_tyNtParamCurr.tyProdRcpMtrPshrExtTorq.diMax/2;
	END_IF
END_ACTION
```

#### Act_OptP0933Navi.st
```iecst
ACTION Act_OptP0933Navi:

	IF tyP0933PullConv.tyNaviBack.tyBtnBack.bRtCompl = TRUE THEN
		tyP0933PullConv.tyNaviBack.tyBtnBack.bRtCompl	:= FALSE;
		tyP0933PullConv.tyNaviBack.tyBtnBack.bValue		:= FALSE;

		eChgPage	:= UIP0920MtrNPneuCtrl;
	END_IF

END_ACTION
```

#### Act_OptP0933FullMask.st
```iecst
ACTION Act_OptP0933FullMask:

	IF eCurrPage = UIP0933PullConv THEN

		IF p_tyDI.bEStopSig = FALSE THEN
			p_tyC0002FullMask ACCESS ADR(tyP0933PullConv.tyFullMaskEStop);

		ELSIF p_tyDI.bCoverSWSig = FALSE THEN
			p_tyC0002FullMask ACCESS ADR(tyP0933PullConv.tyFullMaskCWSig);

		ELSIF p_tyDI.bSafetyRlySig = FALSE THEN
			p_tyC0002FullMask ACCESS ADR(tyP0933PullConv.tyFullMaskSafetyRly);

		ELSIF p_tyNtParamCurr.bAWPrep AND  p_tyNtParamCurr.bAWPusherPrep
			AND p_tyMcParamCurr.bAWDis = FALSE
			AND p_bAWOpenIsHomed = FALSE
			AND (p_diAWPushOrPullerActualPos + p_tyMcParamCurr.diAWPusherAtHmPosInUM )>(p_tyMcParamCurr.diWidthAtHmPosInUM - p_diAWOpenActualPos-15000)
			THEN
			p_tyC0002FullMask ACCESS ADR(tyP0933PullConv.tyFullMaskAWConvInterrupt);

		ELSE
			p_tyC0002FullMask ACCESS ADR(tyP0933PullConv.tyFullMaskHide);

		END_IF

		//Shutter Full mask
		IF p_tyNtParamCurr.bProjInletShutPrep AND p_tyDI.bInShutterOpenRS AND p_tyNtParamCurr.bProjCurtainSenPrep THEN
			IF ABS(p_diTravActualPos - p_diMagRcp1TravPos) > 2500 AND p_tyNtParamCurr.bProjShutter2Prep THEN
				p_tyC0002FullMask ACCESS ADR(tyP0933PullConv.tyFullMaskTravInt);
			END_IF
		ELSIF p_tyNtParamCurr.bProjInletShutPrep AND p_tyDI.bInShutterOpenRS2 THEN
			IF ABS(p_diTravActualPos - p_diMagRcp2TravPos) > 2500 THEN
				p_tyC0002FullMask ACCESS ADR(tyP0933PullConv.tyFullMaskTravInt);//26
			END_IF
		ELSIF p_tyNtParamCurr.bProjInletShutPrep AND p_tyDI.bInShutterOpenRS3 THEN
			IF ABS(p_diTravActualPos - p_diMagRcp3TravPos) > 2500 THEN
				p_tyC0002FullMask ACCESS ADR(tyP0933PullConv.tyFullMaskTravInt);
			END_IF
		ELSIF p_tyNtParamCurr.bProjInletShutPrep AND (p_tyDI.bInShutterOpenRS = FALSE OR  p_tyDI.bInShutterOpenRS2 = FALSE OR p_tyDI.bInShutterOpenRS3 = FALSE) THEN
			IF p_tyNtParamCurr.bProjCurtainSenPrep THEN
				IF (p_tyDI.bInShutterOpenRS = FALSE OR
					(p_tyNtParamCurr.bProjShutter2Prep AND p_tyDI.bInShutterOpenRS2 = FALSE) OR
					(p_tyNtParamCurr.bProjShutter3Prep AND p_tyDI.bInShutterOpenRS3 = FALSE)) THEN
					p_tyC0002FullMask ACCESS ADR(tyP0933PullConv.tyFullMaskInShutterInterrupt); //9
				END_IF
			ELSE //standard
				IF p_tyDI.bInShutterOpenRS = FALSE AND p_tyNtParamCurr.bProjInletShutPrep THEN
					p_tyC0002FullMask ACCESS ADR(tyP0933PullConv.tyFullMaskInShutterInterrupt);
				END_IF
			END_IF
		END_IF //## shutter cond

	END_IF

END_ACTION
```

#### Act_OptP0933Keypad.st
```iecst
ACTION Act_OptP0933Keypad:

	IF fUIOutRtStatTPIsOpen(ADR(tyP0933PullConv.tyFB.tyNumExtSpd.uiRtStat)) = TRUE THEN
		tyProperty.tyKeypad.tyStringTitle.sKeypadTitle	:= tyP0933PullConv.tyFB.tyNumExtSpd.sKeypadTitle;

	ELSIF fUIOutRtStatTPIsOpen(ADR(tyP0933PullConv.tyFB.tyNumExtTorqPercent.uiRtStat)) = TRUE THEN
		tyProperty.tyKeypad.tyStringTitle.sKeypadTitle	:= tyP0933PullConv.tyFB.tyNumExtTorqPercent.sKeypadTitle;

	END_IF

END_ACTION
```

#### Act_OptP0933PullerConvChgLyr.st
```iecst
ACTION Act_OptP0933PullerConvChgLyr:

	IF tyP0933PullConv.tyCom.tyBtnSwitch.bRtCompl THEN
		tyP0933PullConv.tyCom.tyBtnSwitch.bRtCompl := FALSE;

		IF tyP0933PullConv.tyCom.tyBtnSwitch.bValue = TRUE THEN
			fUIInRtStatOff(ADR(tyP0933PullConv.tyDC.tyLyr.uiRtStat));
			fUIInRtStatHide(ADR(tyP0933PullConv.tyFB.tyLyr.uiRtStat));
		ELSE
			fUIInRtStatHide(ADR(tyP0933PullConv.tyDC.tyLyr.uiRtStat));
			fUIInRtStatOff(ADR(tyP0933PullConv.tyFB.tyLyr.uiRtStat));
		END_IF

	END_IF

	//Mask
	IF tyP0933PullConv.tyFB.tyBtnExt.bRtCompl OR tyP0933PullConv.tyFB.tyBtnRet.bRtCompl OR tyP0933PullConv.tyFB.tyBtnStop.bRtCompl
		OR tyP0933PullConv.tyDC.tyBtnAlarmRst.bValue OR tyP0933PullConv.tyDC.tyBtnBrake.bValue OR tyP0933PullConv.tyDC.tyBtnExt.bValue OR tyP0933PullConv.tyDC.tyBtnRet.bValue OR tyP0933PullConv.tyDC.tyBtnSigOn.bValue OR tyP0933PullConv.tyDC.tyBtnSpdBinBit0.bValue OR tyP0933PullConv.tyDC.tyBtnSpdBinBit1.bValue OR tyP0933PullConv.tyDC.tyBtnSpdBinBit2.bValue THEN

		fUIInRtStatOff(ADR(tyP0933PullConv.tyCom.tyBtnSwitch.uiMaskRtStat));
	ELSE
		fUIInRtStatHide(ADR(tyP0933PullConv.tyCom.tyBtnSwitch.uiMaskRtStat));
	END_IF

END_ACTION
```

#### Act_OptP0933PullerConvSen.st
```iecst
ACTION Act_OptP0933PullerConvSen:

	tyP0933PullConv.tyCom.tyBtnLftSen.bValue	:= p_tyDI.bConvLftSen;
	tyP0933PullConv.tyCom.tyBtnRgtSen.bValue	:= p_tyDI.bConvRgtSen;
	tyP0933PullConv.tyCom.tyBtnExtRS.bValue		:= p_tyDI.bPullerExtRS;
	tyP0933PullConv.tyCom.tyBtnRetRS.bValue		:= p_tyDI.bPullerRetRS;
	tyP0933PullConv.tyCom.tyBtnRotHmRS.bValue	:= p_tyDI.bPullerRotHmRS;
	tyP0933PullConv.tyCom.tyBtnRotRmRS.bValue	:= p_tyDI.bPullerRotRmRS;

	tyP0933PullConv.tyCom.tyBtnExtSlwSen.bValue	:= p_tyDI.bPullerExtSlwSen;
	tyP0933PullConv.tyCom.tyBtnRetSlwSen.bValue	:= p_tyDI.bPullerRetSlwSen;

	tyP0933PullConv.tyCom.tyBtnAlarmSig.bValue	:= p_tyDI.bMtrPullerAlmSig;
	tyP0933PullConv.tyCom.tyBtnTorqueSig.bValue	:= p_tyDI.bMtrPullerTorqueSig;
	tyP0933PullConv.tyCom.tyBtnAntiJamSen.bValue := p_tyDI.bPullerAntiJam;
	tyP0933PullConv.tyCom.tyBtnConvClrSen.bValue := p_tyDI.bConvClrSen;

	//Machine Bitmap //8
	IF p_tyNtParamCurr.eProjMag = LDMagTriple AND p_tyNtParamCurr.bMagAutoVerifyPrep = FALSE THEN

		IF tyP0933PullConv.tyFB.tyBtnRotToRm.bRtCompl OR tyP0933PullConv.tyDC.tyBtnRotToRm.bRtCompl THEN
			IF p_tyDI.bPullerExtRS = TRUE THEN
				tyP0933PullConv.tyCom.tyBitmapMc.uiValueIdx	:= 4; //ext rm //12
			ELSE
				tyP0933PullConv.tyCom.tyBitmapMc.uiValueIdx	:= 2; //ret //10
			END_IF

		ELSIF tyP0933PullConv.tyFB.tyBtnRotToHm.bRtCompl OR tyP0933PullConv.tyDC.tyBtnRotToHm.bRtCompl THEN
			IF p_tyDI.bPullerExtRS = TRUE THEN
				tyP0933PullConv.tyCom.tyBitmapMc.uiValueIdx	:= 3; //ext hm //11
			ELSE
				tyP0933PullConv.tyCom.tyBitmapMc.uiValueIdx	:= 1; //9
			END_IF

		ELSIF tyP0933PullConv.tyFB.tyBtnExt.bRtCompl OR tyP0933PullConv.tyDC.tyBtnExt.bRtCompl THEN
			IF p_tyDI.bPullerRotRmRS = TRUE THEN
				tyP0933PullConv.tyCom.tyBitmapMc.uiValueIdx	:= 4; //ext//12
			ELSE
				tyP0933PullConv.tyCom.tyBitmapMc.uiValueIdx	:= 3; //11
			END_IF

		ELSIF tyP0933PullConv.tyFB.tyBtnRet.bRtCompl OR tyP0933PullConv.tyDC.tyBtnRet.bRtCompl THEN
			IF p_tyDI.bPullerRotRmRS = TRUE THEN
				tyP0933PullConv.tyCom.tyBitmapMc.uiValueIdx	:= 2; //10
			ELSE
				tyP0933PullConv.tyCom.tyBitmapMc.uiValueIdx	:= 1; //9
			END_IF

		ELSIF tyP0933PullConv.tyFB.tyBtnCylEnt.bRtCompl OR tyP0933PullConv.tyFB.tyBtnEnt.bRtCompl OR tyP0933PullConv.tyFB.tyBtnExit.bRtCompl OR tyP0933PullConv.tyFB.tyBtnStop.bRtCompl
			OR tyP0933PullConv.tyDC.tyBtnStart.bRtCompl OR tyP0933PullConv.tyDC.tyBtnStop.bRtCompl THEN

			tyP0933PullConv.tyCom.tyBitmapMc.uiValueIdx	:= 0; //8

		END_IF

		IF p_tyNtParamCurr.bProjMotorizedPullerPrep = FALSE THEN
			IF	tyP0933PullConv.tyCom.tyBitmapMc.uiValueIdx < 200 AND  p_tyNtParamCurr.bProjTopToBtmDefault = TRUE  THEN
				tyP0933PullConv.tyCom.tyBitmapMc.uiValueIdx	:= tyP0933PullConv.tyCom.tyBitmapMc.uiValueIdx + 200;
			END_IF
			IF tyP0933PullConv.tyCom.tyBitmapMc.uiValueIdx < 108-8 AND  p_tyNtParamCurr.bProjTopToBtmDefault = FALSE  THEN
				tyP0933PullConv.tyCom.tyBitmapMc.uiValueIdx	:= tyP0933PullConv.tyCom.tyBitmapMc.uiValueIdx + 108-8;
			END_IF
		ELSIF p_tyNtParamCurr.bProjMotorizedPullerPrep = TRUE AND p_tyNtParamCurr.bProjPullerRotCylPrep = FALSE THEN //fix (siemens)
			IF	tyP0933PullConv.tyCom.tyBitmapMc.uiValueIdx < 389-8 THEN
				tyP0933PullConv.tyCom.tyBitmapMc.uiValueIdx	:= tyP0933PullConv.tyCom.tyBitmapMc.uiValueIdx + 389-8;
			END_IF
		ELSIF p_tyNtParamCurr.bProjMotorizedPullerPrep = TRUE AND p_tyNtParamCurr.bProjCurtainSenPrep = FALSE THEN
			IF	tyP0933PullConv.tyCom.tyBitmapMc.uiValueIdx < 300 THEN
				tyP0933PullConv.tyCom.tyBitmapMc.uiValueIdx	:= tyP0933PullConv.tyCom.tyBitmapMc.uiValueIdx + 300;
			END_IF
		ELSIF p_tyNtParamCurr.bProjMotorizedPullerPrep = TRUE AND p_tyNtParamCurr.bProjCurtainSenPrep AND p_tyNtParamCurr.bProjTopToBtmDefault = TRUE THEN
			IF	tyP0933PullConv.tyCom.tyBitmapMc.uiValueIdx < 379-8 THEN
				tyP0933PullConv.tyCom.tyBitmapMc.uiValueIdx	:= tyP0933PullConv.tyCom.tyBitmapMc.uiValueIdx + 379-8;
			END_IF
		ELSIF p_tyNtParamCurr.bProjMotorizedPullerPrep = TRUE AND p_tyNtParamCurr.bProjCurtainSenPrep = TRUE AND p_tyNtParamCurr.bProjTopToBtmDefault = FALSE  THEN
			IF	tyP0933PullConv.tyCom.tyBitmapMc.uiValueIdx < 430-8 THEN
				tyP0933PullConv.tyCom.tyBitmapMc.uiValueIdx	:= tyP0933PullConv.tyCom.tyBitmapMc.uiValueIdx + 430-8;
			END_IF
		END_IF

	ELSIF p_tyNtParamCurr.eProjMag = LDMagDual AND p_tyNtParamCurr.bMagAutoVerifyPrep = FALSE THEN

		IF tyP0933PullConv.tyFB.tyBtnRotToRm.bRtCompl OR tyP0933PullConv.tyDC.tyBtnRotToRm.bRtCompl THEN
			IF p_tyDI.bPullerExtRS = TRUE THEN
				tyP0933PullConv.tyCom.tyBitmapMc.uiValueIdx	:= 4; //ext rm //12
			ELSE
				tyP0933PullConv.tyCom.tyBitmapMc.uiValueIdx	:= 2; //ret //10
			END_IF

		ELSIF tyP0933PullConv.tyFB.tyBtnRotToHm.bRtCompl OR tyP0933PullConv.tyDC.tyBtnRotToHm.bRtCompl THEN
			IF p_tyDI.bPullerExtRS = TRUE THEN
				tyP0933PullConv.tyCom.tyBitmapMc.uiValueIdx	:= 3; //ext hm //11
			ELSE
				tyP0933PullConv.tyCom.tyBitmapMc.uiValueIdx	:= 1; //9
			END_IF

		ELSIF tyP0933PullConv.tyFB.tyBtnExt.bRtCompl OR tyP0933PullConv.tyDC.tyBtnExt.bRtCompl THEN
			IF p_tyDI.bPullerRotRmRS = TRUE THEN
				tyP0933PullConv.tyCom.tyBitmapMc.uiValueIdx	:= 4; //ext//12
			ELSE
				tyP0933PullConv.tyCom.tyBitmapMc.uiValueIdx	:= 3; //11
			END_IF

		ELSIF tyP0933PullConv.tyFB.tyBtnRet.bRtCompl OR tyP0933PullConv.tyDC.tyBtnRet.bRtCompl THEN
			IF p_tyDI.bPullerRotRmRS = TRUE THEN
				tyP0933PullConv.tyCom.tyBitmapMc.uiValueIdx	:= 2; //10
			ELSE
				tyP0933PullConv.tyCom.tyBitmapMc.uiValueIdx	:= 1; //9
			END_IF

		ELSIF tyP0933PullConv.tyFB.tyBtnCylEnt.bRtCompl OR tyP0933PullConv.tyFB.tyBtnEnt.bRtCompl OR tyP0933PullConv.tyFB.tyBtnExit.bRtCompl OR tyP0933PullConv.tyFB.tyBtnStop.bRtCompl
			OR tyP0933PullConv.tyDC.tyBtnStart.bRtCompl OR tyP0933PullConv.tyDC.tyBtnStop.bRtCompl THEN

			tyP0933PullConv.tyCom.tyBitmapMc.uiValueIdx	:= 0; //8

		END_IF

		IF p_tyNtParamCurr.bProjMotorizedPullerPrep = FALSE THEN
			IF	tyP0933PullConv.tyCom.tyBitmapMc.uiValueIdx < 200 AND  p_tyNtParamCurr.bProjTopToBtmDefault = TRUE AND p_tyNtParamCurr.bUIConvDirRL THEN
				tyP0933PullConv.tyCom.tyBitmapMc.uiValueIdx	:= tyP0933PullConv.tyCom.tyBitmapMc.uiValueIdx + 488-8;
			END_IF
		ELSIF p_tyNtParamCurr.bProjMotorizedPullerPrep THEN
			IF	tyP0933PullConv.tyCom.tyBitmapMc.uiValueIdx < 200 AND  p_tyNtParamCurr.bProjTopToBtmDefault = TRUE AND p_tyNtParamCurr.bUIConvDirRL THEN
				tyP0933PullConv.tyCom.tyBitmapMc.uiValueIdx	:= tyP0933PullConv.tyCom.tyBitmapMc.uiValueIdx + 458-8;
			END_IF
		END_IF
//	ELSIF p_tyNtParamCurr.eProjMag = LDMagDual AND p_tyNtParamCurr.bMagAutoVerifyPrep = FALSE THEN
//
//		IF tyP0933PullConv.tyFB.tyBtnRotToRm.bRtCompl OR tyP0933PullConv.tyDC.tyBtnRotToRm.bRtCompl THEN
//
//			tyP0933PullConv.tyCom.tyBitmapMc.uiValueIdx	:= 4;//== 2
//
//		ELSIF tyP0933PullConv.tyFB.tyBtnRotToHm.bRtCompl OR tyP0933PullConv.tyDC.tyBtnRotToHm.bRtCompl THEN
//			IF p_tyDI.bPullerExtRS THEN
//				tyP0933PullConv.tyCom.tyBitmapMc.uiValueIdx	:= 2;
//			ELSIF p_tyDI.bPullerRetRS THEN
//				tyP0933PullConv.tyCom.tyBitmapMc.uiValueIdx	:= 1;
//			END_IF
//			//tyP0933PullConv.tyCom.tyBitmapMc.uiValueIdx	:= 3;
//
//		ELSIF tyP0933PullConv.tyFB.tyBtnExt.bRtCompl OR tyP0933PullConv.tyDC.tyBtnExt.bRtCompl THEN
//
//			tyP0933PullConv.tyCom.tyBitmapMc.uiValueIdx	:= 2;
//
//		ELSIF tyP0933PullConv.tyFB.tyBtnRet.bRtCompl OR tyP0933PullConv.tyDC.tyBtnRet.bRtCompl THEN
//
//			tyP0933PullConv.tyCom.tyBitmapMc.uiValueIdx	:= 1;
//
//		ELSIF tyP0933PullConv.tyFB.tyBtnCylEnt.bRtCompl OR tyP0933PullConv.tyFB.tyBtnEnt.bRtCompl OR tyP0933PullConv.tyFB.tyBtnExit.bRtCompl OR tyP0933PullConv.tyFB.tyBtnStop.bRtCompl
//			OR tyP0933PullConv.tyDC.tyBtnStart.bRtCompl OR tyP0933PullConv.tyDC.tyBtnStop.bRtCompl THEN
//
//			tyP0933PullConv.tyCom.tyBitmapMc.uiValueIdx	:= 0;
//
//		END_IF
//
//
//		IF tyP0933PullConv.tyCom.tyBitmapMc.uiValueIdx < 200 THEN
//			tyP0933PullConv.tyCom.tyBitmapMc.uiValueIdx	:= tyP0933PullConv.tyCom.tyBitmapMc.uiValueIdx + 200;
//		END_IF

	ELSIF p_tyNtParamCurr.bMagAutoVerifyPrep = TRUE THEN

	//		IF tyP0933PullConv.tyFB.tyBtnRotToRm.bRtCompl OR tyP0933PullConv.tyDC.tyBtnRotToRm.bRtCompl THEN
	//
	//			IF p_tyDI.bPullerExtRS = TRUE THEN
	//				tyP0933PullConv.tyCom.tyBitmapMc.uiValueIdx	:= 4;
	//			ELSE
	//				tyP0933PullConv.tyCom.tyBitmapMc.uiValueIdx	:= 2;
	//			END_IF
	//
	//		ELSIF tyP0933PullConv.tyFB.tyBtnRotToHm.bRtCompl OR tyP0933PullConv.tyDC.tyBtnRotToHm.bRtCompl THEN
	//
	//			IF p_tyDI.bPullerExtRS = TRUE THEN
	//				tyP0933PullConv.tyCom.tyBitmapMc.uiValueIdx	:= 3;
	//			ELSE
	//				tyP0933PullConv.tyCom.tyBitmapMc.uiValueIdx	:= 1;
	//			END_IF
	//
	//		ELSIF tyP0933PullConv.tyFB.tyBtnExt.bRtCompl OR tyP0933PullConv.tyDC.tyBtnExt.bRtCompl THEN
	//
	//			IF p_tyDI.bPullerRotRmRS = TRUE THEN
	//				tyP0933PullConv.tyCom.tyBitmapMc.uiValueIdx	:= 4;
	//			ELSE
	//				tyP0933PullConv.tyCom.tyBitmapMc.uiValueIdx	:= 3;
	//			END_IF
	//
	//		ELSIF tyP0933PullConv.tyFB.tyBtnRet.bRtCompl OR tyP0933PullConv.tyDC.tyBtnRet.bRtCompl THEN
	//
	//			IF p_tyDI.bPullerRotRmRS = TRUE THEN
	//				tyP0933PullConv.tyCom.tyBitmapMc.uiValueIdx	:= 2;
	//			ELSE
	//				tyP0933PullConv.tyCom.tyBitmapMc.uiValueIdx	:= 1;
	//			END_IF

		IF tyP0933PullConv.tyFB.tyBtnRotToRm.bRtCompl OR tyP0933PullConv.tyDC.tyBtnRotToRm.bRtCompl THEN

			tyP0933PullConv.tyCom.tyBitmapMc.uiValueIdx	:= 0;

		ELSIF tyP0933PullConv.tyFB.tyBtnRotToHm.bRtCompl OR tyP0933PullConv.tyDC.tyBtnRotToHm.bRtCompl THEN

			tyP0933PullConv.tyCom.tyBitmapMc.uiValueIdx	:= 0;

		ELSIF tyP0933PullConv.tyFB.tyBtnExt.bRtCompl OR tyP0933PullConv.tyDC.tyBtnExt.bRtCompl THEN

			tyP0933PullConv.tyCom.tyBitmapMc.uiValueIdx	:= 0;

		ELSIF tyP0933PullConv.tyFB.tyBtnRet.bRtCompl OR tyP0933PullConv.tyDC.tyBtnRet.bRtCompl THEN

			tyP0933PullConv.tyCom.tyBitmapMc.uiValueIdx	:= 0;

		ELSIF tyP0933PullConv.tyFB.tyBtnCylEnt.bRtCompl OR tyP0933PullConv.tyFB.tyBtnEnt.bRtCompl OR tyP0933PullConv.tyFB.tyBtnExit.bRtCompl OR tyP0933PullConv.tyFB.tyBtnStop.bRtCompl
			OR tyP0933PullConv.tyDC.tyBtnStart.bRtCompl OR tyP0933PullConv.tyDC.tyBtnStop.bRtCompl THEN

			tyP0933PullConv.tyCom.tyBitmapMc.uiValueIdx	:= 0;

		END_IF

		IF tyP0933PullConv.tyCom.tyBitmapMc.uiValueIdx < 200 THEN
			tyP0933PullConv.tyCom.tyBitmapMc.uiValueIdx	:= tyP0933PullConv.tyCom.tyBitmapMc.uiValueIdx + 200;
		END_IF

	END_IF
END_ACTION
```

#### Act_OptP0933PullerConvFB.st
```iecst
ACTION Act_OptP0933PullerConvFB:

	//Parameter
	diMnlMtrPshrExtSpd	:= tyP0933PullConv.tyFB.tyNumExtSpd.diValue;
	//diMnlMtrPshrExtTorq	:= tyP0933PullConv.tyFB.tyNumExtTorqPercent.diValue;
//	diMnlMtrPshrExtTorq	:= 30 + ((72/90)*(tyP0933PullConv.tyFB.tyNumExtTorqPercent.diValue - 10)); //70 = 100N -30N
//	diMnlMtrPshrExtTorq := 15 + (((tyP0933PullConv.tyFB.tyNumExtTorqPercent.diValue -10)/10)*167/100); //15-30 N used
//	diMnlMtrPshrExtTorq := p_tyNtParamCurr.tyPPTorqParam.usiStartTorque + (((tyP0933PullConv.tyFB.tyNumExtTorqPercent.diValue -10)/10)*p_tyNtParamCurr.tyPPTorqParam.uiRatio/100); //17-50 N used
	diMnlMtrPshrExtTorq := p_tyNtParamCurr.tyPPTorqParam.usiStartTorque + REAL_TO_DINT(DINT_TO_REAL(tyP0933PullConv.tyFB.tyNumExtTorqPercent.diValue -10)*UINT_TO_REAL(p_tyNtParamCurr.tyPPTorqParam.uiRatio)/1000.0);
	//Alarm
	IF p_bAlarmErr THEN
		tyP0933PullConv.tyFB.tyBtnStop.bRtCompl := TRUE;
	END_IF

	//Conveyor
	IF tyP0933PullConv.tyFB.tyBtnStop.bRtCompl = TRUE THEN
		diMnlPPJogSpd	:= 0;
		ePullConvAct	:= ConvActPullerRstAll;

		IF  p_ePullConvStat = ConvActPullerRstAll AND p_ePullConvStatus = Done THEN

			ePullConvAct	:= ConvActIdle;

			tyP0933PullConv.tyFB.tyBtnCylEnt.bRtCompl	:= FALSE;
			tyP0933PullConv.tyFB.tyBtnCylEnt.bValue		:= FALSE;
			tyP0933PullConv.tyFB.tyBtnCylEnt.bRtLk		:= FALSE;

			tyP0933PullConv.tyFB.tyBtnEnt.bRtCompl		:= FALSE;
			tyP0933PullConv.tyFB.tyBtnEnt.bValue		:= FALSE;
			tyP0933PullConv.tyFB.tyBtnEnt.bRtLk			:= FALSE;

			tyP0933PullConv.tyFB.tyBtnExit.bRtCompl		:= FALSE;
			tyP0933PullConv.tyFB.tyBtnExit.bValue		:= FALSE;
			tyP0933PullConv.tyFB.tyBtnExit.bRtLk		:= FALSE;

			tyP0933PullConv.tyFB.tyBtnStop.bRtCompl		:= FALSE;
			tyP0933PullConv.tyFB.tyBtnStop.bValue		:= TRUE;
			tyP0933PullConv.tyFB.tyBtnStop.bRtLk		:= TRUE;
		END_IF

	ELSIF tyP0933PullConv.tyFB.tyBtnCylEnt.bRtCompl = TRUE THEN
		tyP0933PullConv.tyFB.tyBtnCylEnt.bValue		:= TRUE;
		tyP0933PullConv.tyFB.tyBtnCylEnt.bRtLk		:= TRUE;

		tyP0933PullConv.tyFB.tyBtnStop.bValue		:= FALSE;
		tyP0933PullConv.tyFB.tyBtnStop.bRtLk		:= FALSE;
		diMnlPPJogSpd	:= diMnlMtrPshrExtSpd*diMnlServoMtrMaxPulRatio;
		ePullConvAct	:= ConvActEntPuller;

		fUIInRtStatOff(ADR(tyP0933PullConv.tyCom.tyBtnSwitch.uiMaskRtStat));

		IF p_ePullConvStat = ConvActEntPuller AND p_ePullConvStatus = Done THEN
			ePullConvAct	:= ConvActIdle;

			tyP0933PullConv.tyFB.tyBtnCylEnt.bRtCompl	:= FALSE;

			tyP0933PullConv.tyFB.tyBtnCylEnt.bValue		:= FALSE;
			tyP0933PullConv.tyFB.tyBtnCylEnt.bRtLk		:= FALSE;

			tyP0933PullConv.tyFB.tyBtnStop.bValue		:= FALSE;
			tyP0933PullConv.tyFB.tyBtnStop.bRtLk		:= FALSE;

		fUIInRtStatHide(ADR(tyP0933PullConv.tyCom.tyBtnSwitch.uiMaskRtStat));

		END_IF

	ELSIF tyP0933PullConv.tyFB.tyBtnEnt.bRtCompl = TRUE THEN
		tyP0933PullConv.tyFB.tyBtnEnt.bValue	:= TRUE;
		tyP0933PullConv.tyFB.tyBtnEnt.bRtLk		:= TRUE;

		tyP0933PullConv.tyFB.tyBtnStop.bValue	:= FALSE;
		tyP0933PullConv.tyFB.tyBtnStop.bRtLk	:= FALSE;

		ePullConvAct	:= ConvActEnt;
		fUIInRtStatOff(ADR(tyP0930MagConv1.tyCom.tyBtnSwitch.uiMaskRtStat));

		IF p_ePullConvStat = ConvActEnt AND p_ePullConvStatus = Done THEN
			ePullConvAct	:= ConvActIdle;

			tyP0933PullConv.tyFB.tyBtnEnt.bRtCompl	:= FALSE;

			tyP0933PullConv.tyFB.tyBtnEnt.bValue	:= FALSE;
			tyP0933PullConv.tyFB.tyBtnEnt.bRtLk		:= FALSE;

			tyP0933PullConv.tyFB.tyBtnStop.bValue	:= FALSE;
			tyP0933PullConv.tyFB.tyBtnStop.bRtLk	:= FALSE;

			fUIInRtStatHide(ADR(tyP0930MagConv1.tyCom.tyBtnSwitch.uiMaskRtStat));
		END_IF

	ELSIF tyP0933PullConv.tyFB.tyBtnExit.bRtCompl = TRUE THEN
		tyP0933PullConv.tyFB.tyBtnExit.bValue	:= TRUE;
		tyP0933PullConv.tyFB.tyBtnExit.bRtLk	:= TRUE;

		tyP0933PullConv.tyFB.tyBtnStop.bValue	:= FALSE;
		tyP0933PullConv.tyFB.tyBtnStop.bRtLk	:= FALSE;

		ePullConvAct	:= ConvActExit;

		fUIInRtStatOff(ADR(tyP0930MagConv1.tyCom.tyBtnSwitch.uiMaskRtStat));

		IF p_ePullConvStat = ConvActExit AND p_ePullConvStatus = Done THEN
			ePullConvAct	:= ConvActIdle;

			tyP0933PullConv.tyFB.tyBtnExit.bRtCompl	:= FALSE;

			tyP0933PullConv.tyFB.tyBtnExit.bValue	:= FALSE;
			tyP0933PullConv.tyFB.tyBtnExit.bRtLk	:= FALSE;

			tyP0933PullConv.tyFB.tyBtnStop.bValue	:= FALSE;
			tyP0933PullConv.tyFB.tyBtnStop.bRtLk	:= FALSE;

			fUIInRtStatHide(ADR(tyP0930MagConv1.tyCom.tyBtnSwitch.uiMaskRtStat));
		END_IF

	END_IF

	//Puller
	IF (p_tyNtParamCurr.bProjPullerRotCylPrep = TRUE OR p_tyNtParamCurr.bProjMotorizedPullerPrep) AND tyP0933PullConv.tyFB.tyBtnStop.bRtCompl = FALSE THEN

		IF tyP0933PullConv.tyCom.tyBtnSwitch.bValue = FALSE THEN
			IF tyP0933PullConv.tyFB.tyBtnRet.bRtCompl = TRUE THEN
				tyP0933PullConv.tyFB.tyBtnRet.bRtCompl	:= FALSE;

				tyP0933PullConv.tyFB.tyBtnRet.bValue	:= TRUE;
				tyP0933PullConv.tyFB.tyBtnExt.bValue	:= FALSE;

			ELSIF tyP0933PullConv.tyFB.tyBtnExt.bRtCompl = TRUE THEN
				tyP0933PullConv.tyFB.tyBtnExt.bRtCompl	:= FALSE;

				tyP0933PullConv.tyFB.tyBtnExt.bValue	:= TRUE;
				tyP0933PullConv.tyFB.tyBtnRet.bValue	:= FALSE;

			END_IF

			IF tyP0933PullConv.tyFB.tyBtnRet.bValue = TRUE THEN
				ePullConvAct	:= ConvActPullerRet;
				diMnlPPJogSpd	:= diMnlMtrPshrExtSpd*diMnlServoMtrMaxPulRatio;

				tyP0933PullConv.tyFB.tyBtnStop.bValue		:= FALSE;
				tyP0933PullConv.tyFB.tyBtnStop.bRtLk		:= FALSE;

				IF p_ePullConvStat = ConvActPullerRet AND p_ePullConvStatus = Done THEN
					ePullConvAct	:= ConvActIdle;
					diMnlPPJogSpd	:= 0;
					tyP0933PullConv.tyFB.tyBtnRet.bValue	:= FALSE;

				ELSIF p_ePullConvStatus = Error THEN
					tyP0933PullConv.tyFB.tyBtnRet.bValue	:= FALSE;
					diMnlPPJogSpd	:= 0;
				END_IF

			ELSIF tyP0933PullConv.tyFB.tyBtnExt.bValue = TRUE THEN
				ePullConvAct	:= ConvActPullerExt;
				diMnlPPJogSpd	:= diMnlMtrPshrExtSpd*diMnlServoMtrMaxPulRatio;
				tyP0933PullConv.tyFB.tyBtnStop.bValue		:= FALSE;
				tyP0933PullConv.tyFB.tyBtnStop.bRtLk		:= FALSE;

				IF p_ePullConvStat = ConvActPullerExt AND p_ePullConvStatus = Done THEN
					ePullConvAct	:= ConvActIdle;
					diMnlPPJogSpd	:= 0;
					tyP0933PullConv.tyFB.tyBtnExt.bValue := FALSE;

				ELSIF p_ePullConvStatus = Error THEN
					tyP0933PullConv.tyFB.tyBtnExt.bValue := FALSE;
					diMnlPPJogSpd	:= 0;
				END_IF

			END_IF

			//Update Status
			tyP0933PullConv.tyDC.tyBtnRet.bValue	:= p_bPullConvPullerRetCtrl;
			tyP0933PullConv.tyDC.tyBtnExt.bValue	:= p_bPullConvPullerExtCtrl;

		END_IF

	ELSIF p_tyNtParamCurr.bProjPullerRotCylPrep = FALSE AND tyP0933PullConv.tyFB.tyBtnStop.bRtCompl = FALSE
		THEN

		IF tyP0933PullConv.tyCom.tyBtnSwitch.bValue = FALSE THEN
			IF tyP0933PullConv.tyFB.tyBtnRet.bRtCompl = TRUE THEN
				tyP0933PullConv.tyFB.tyBtnRet.bRtCompl	:= FALSE;

				tyP0933PullConv.tyFB.tyBtnRet.bValue	:= TRUE;
				tyP0933PullConv.tyFB.tyBtnExt.bValue	:= FALSE;

			ELSIF tyP0933PullConv.tyFB.tyBtnExt.bRtCompl = TRUE THEN
				tyP0933PullConv.tyFB.tyBtnExt.bRtCompl	:= FALSE;

				tyP0933PullConv.tyFB.tyBtnExt.bValue	:= TRUE;
				tyP0933PullConv.tyFB.tyBtnRet.bValue	:= FALSE;

			END_IF

			IF tyP0933PullConv.tyFB.tyBtnRet.bValue = TRUE THEN
				ePullerAct	:= PneuActRet;

				tyP0933PullConv.tyFB.tyBtnStop.bValue		:= FALSE;
				tyP0933PullConv.tyFB.tyBtnStop.bRtLk		:= FALSE;

				IF p_ePullerStat = PneuActRet AND p_ePullerStatus = Done THEN
					ePullerAct	:= PneuActIdle;

					tyP0933PullConv.tyFB.tyBtnRet.bValue	:= FALSE;

				ELSIF p_ePullerStatus = Error THEN
					tyP0933PullConv.tyFB.tyBtnRet.bValue	:= FALSE;

				END_IF

			ELSIF tyP0933PullConv.tyFB.tyBtnExt.bValue = TRUE THEN
				ePullerAct	:= PneuActExt;

				tyP0933PullConv.tyFB.tyBtnStop.bValue		:= FALSE;
				tyP0933PullConv.tyFB.tyBtnStop.bRtLk		:= FALSE;

				IF p_ePullerStat = PneuActExt AND p_ePullerStatus = Done THEN
					ePullerAct	:= PneuActIdle;

					tyP0933PullConv.tyFB.tyBtnExt.bValue := FALSE;

				ELSIF p_ePullerStatus = Error THEN
					tyP0933PullConv.tyFB.tyBtnExt.bValue := FALSE;

				END_IF

			END_IF

			//Update Status
			tyP0933PullConv.tyDC.tyBtnRet.bValue	:= p_bPullerRetCtrl;
			tyP0933PullConv.tyDC.tyBtnExt.bValue	:= p_bPullerExtCtrl;

		END_IF

	ELSE

		tyP0933PullConv.tyFB.tyBtnExt.bRtCompl		:= FALSE;
		tyP0933PullConv.tyFB.tyBtnExt.bValue		:= FALSE;
		tyP0933PullConv.tyFB.tyBtnExt.bRtLk			:= FALSE;

		tyP0933PullConv.tyFB.tyBtnRet.bRtCompl		:= FALSE;
		tyP0933PullConv.tyFB.tyBtnRet.bValue		:= FALSE;
		tyP0933PullConv.tyFB.tyBtnRet.bRtLk			:= FALSE;

	END_IF

	//Rotating Cylinder
	IF tyP0933PullConv.tyCom.tyBtnSwitch.bValue = FALSE THEN
		IF tyP0933PullConv.tyFB.tyBtnRotToHm.bRtCompl = TRUE THEN
			tyP0933PullConv.tyFB.tyBtnRotToHm.bRtCompl	:= FALSE;

			tyP0933PullConv.tyFB.tyBtnRotToHm.bValue	:= TRUE;
			tyP0933PullConv.tyFB.tyBtnRotToRm.bValue	:= FALSE;

		ELSIF tyP0933PullConv.tyFB.tyBtnRotToRm.bRtCompl = TRUE THEN
			tyP0933PullConv.tyFB.tyBtnRotToRm.bRtCompl	:= FALSE;

			tyP0933PullConv.tyFB.tyBtnRotToRm.bValue	:= TRUE;
			tyP0933PullConv.tyFB.tyBtnRotToHm.bValue	:= FALSE;

		END_IF

		IF tyP0933PullConv.tyFB.tyBtnRotToHm.bValue = TRUE THEN
			ePullConvAct	:= ConvActRotHome;

			IF p_ePullConvStat = ConvActRotHome AND p_ePullConvStatus = Done THEN
				ePullConvAct	:= ConvActIdle;

				tyP0933PullConv.tyFB.tyBtnRotToHm.bValue	:= FALSE;

			ELSIF p_ePullConvStatus = Error THEN
				tyP0933PullConv.tyFB.tyBtnRotToHm.bValue	:= FALSE;

			END_IF

		ELSIF tyP0933PullConv.tyFB.tyBtnRotToRm.bValue = TRUE THEN
			ePullConvAct	:= ConvActRotRemote;

			IF p_ePullConvStat = ConvActRotRemote AND p_ePullConvStatus = Done THEN
				ePullConvAct	:= ConvActIdle;

				tyP0933PullConv.tyFB.tyBtnRotToRm.bValue := FALSE;

			ELSIF p_ePullConvStatus = Error THEN
				tyP0933PullConv.tyFB.tyBtnRotToRm.bValue := FALSE;

			END_IF

		END_IF

		//Update Status
		tyP0933PullConv.tyDC.tyBtnRotToHm.bValue	:= NOT p_bPullConvRotRemoteCtrl;
		tyP0933PullConv.tyDC.tyBtnRotToRm.bValue	:= p_bPullConvRotRemoteCtrl;

	END_IF

	//Mask
	IF p_tyUsrMgmtCurrAccessRgt.bManualFBOnly THEN

		fUIInRtStatOff(ADR(tyP0933PullConv.tyCom.tyBtnSwitch.uiMaskRtStat));
	ELSE

		IF p_ePullConvStatus = Error THEN

			fUIInRtStatOff(ADR(tyP0933PullConv.tyFB.tyBtnCylEnt.uiMaskRtStat));
			fUIInRtStatOff(ADR(tyP0933PullConv.tyFB.tyBtnEnt.uiMaskRtStat));
			fUIInRtStatOff(ADR(tyP0933PullConv.tyFB.tyBtnExit.uiMaskRtStat));
			fUIInRtStatOff(ADR(tyP0933PullConv.tyFB.tyBtnExt.uiMaskRtStat));
			fUIInRtStatOff(ADR(tyP0933PullConv.tyFB.tyBtnRet.uiMaskRtStat));
			fUIInRtStatOff(ADR(tyP0933PullConv.tyFB.tyBtnRotToHm.uiMaskRtStat));
			fUIInRtStatOff(ADR(tyP0933PullConv.tyFB.tyBtnRotToRm.uiMaskRtStat));
			fUIInRtStatHide(ADR(tyP0933PullConv.tyCom.tyBtnSwitch.uiMaskRtStat));

		ELSIF tyP0933PullConv.tyFB.tyBtnCylEnt.bRtCompl = TRUE THEN

			fUIInRtStatHide(ADR(tyP0933PullConv.tyFB.tyBtnCylEnt.uiMaskRtStat));
			fUIInRtStatOff(ADR(tyP0933PullConv.tyFB.tyBtnEnt.uiMaskRtStat));
			fUIInRtStatOff(ADR(tyP0933PullConv.tyFB.tyBtnExit.uiMaskRtStat));
			fUIInRtStatOff(ADR(tyP0933PullConv.tyFB.tyBtnExt.uiMaskRtStat));
			fUIInRtStatOff(ADR(tyP0933PullConv.tyFB.tyBtnRet.uiMaskRtStat));
			fUIInRtStatOff(ADR(tyP0933PullConv.tyFB.tyBtnRotToHm.uiMaskRtStat));
			fUIInRtStatOff(ADR(tyP0933PullConv.tyFB.tyBtnRotToRm.uiMaskRtStat));
			fUIInRtStatOff(ADR(tyP0933PullConv.tyCom.tyBtnSwitch.uiMaskRtStat));

		ELSIF tyP0933PullConv.tyFB.tyBtnEnt.bRtCompl = TRUE THEN

			fUIInRtStatOff(ADR(tyP0933PullConv.tyFB.tyBtnCylEnt.uiMaskRtStat));
			fUIInRtStatHide(ADR(tyP0933PullConv.tyFB.tyBtnEnt.uiMaskRtStat));
			fUIInRtStatOff(ADR(tyP0933PullConv.tyFB.tyBtnExit.uiMaskRtStat));
			fUIInRtStatOff(ADR(tyP0933PullConv.tyFB.tyBtnExt.uiMaskRtStat));
			fUIInRtStatOff(ADR(tyP0933PullConv.tyFB.tyBtnRet.uiMaskRtStat));
			fUIInRtStatOff(ADR(tyP0933PullConv.tyFB.tyBtnRotToHm.uiMaskRtStat));
			fUIInRtStatOff(ADR(tyP0933PullConv.tyFB.tyBtnRotToRm.uiMaskRtStat));
			fUIInRtStatOff(ADR(tyP0933PullConv.tyCom.tyBtnSwitch.uiMaskRtStat));

		ELSIF tyP0933PullConv.tyFB.tyBtnExit.bRtCompl = TRUE THEN

			fUIInRtStatOff(ADR(tyP0933PullConv.tyFB.tyBtnCylEnt.uiMaskRtStat));
			fUIInRtStatOff(ADR(tyP0933PullConv.tyFB.tyBtnEnt.uiMaskRtStat));
			fUIInRtStatHide(ADR(tyP0933PullConv.tyFB.tyBtnExit.uiMaskRtStat));
			fUIInRtStatOff(ADR(tyP0933PullConv.tyFB.tyBtnExt.uiMaskRtStat));
			fUIInRtStatOff(ADR(tyP0933PullConv.tyFB.tyBtnRet.uiMaskRtStat));
			fUIInRtStatOff(ADR(tyP0933PullConv.tyFB.tyBtnRotToHm.uiMaskRtStat));
			fUIInRtStatOff(ADR(tyP0933PullConv.tyFB.tyBtnRotToRm.uiMaskRtStat));
			fUIInRtStatOff(ADR(tyP0933PullConv.tyCom.tyBtnSwitch.uiMaskRtStat));

		ELSIF tyP0933PullConv.tyFB.tyBtnExt.bValue = TRUE OR tyP0933PullConv.tyFB.tyBtnRet.bValue = TRUE THEN

			fUIInRtStatOff(ADR(tyP0933PullConv.tyFB.tyBtnCylEnt.uiMaskRtStat));
			fUIInRtStatOff(ADR(tyP0933PullConv.tyFB.tyBtnEnt.uiMaskRtStat));
			fUIInRtStatOff(ADR(tyP0933PullConv.tyFB.tyBtnExit.uiMaskRtStat));
			fUIInRtStatHide(ADR(tyP0933PullConv.tyFB.tyBtnExt.uiMaskRtStat));
			fUIInRtStatHide(ADR(tyP0933PullConv.tyFB.tyBtnRet.uiMaskRtStat));
			fUIInRtStatOff(ADR(tyP0933PullConv.tyFB.tyBtnRotToHm.uiMaskRtStat));
			fUIInRtStatOff(ADR(tyP0933PullConv.tyFB.tyBtnRotToRm.uiMaskRtStat));
			fUIInRtStatOff(ADR(tyP0933PullConv.tyCom.tyBtnSwitch.uiMaskRtStat));

		ELSIF tyP0933PullConv.tyFB.tyBtnRotToHm.bValue = TRUE OR tyP0933PullConv.tyFB.tyBtnRotToRm.bValue = TRUE THEN

			fUIInRtStatOff(ADR(tyP0933PullConv.tyFB.tyBtnCylEnt.uiMaskRtStat));
			fUIInRtStatOff(ADR(tyP0933PullConv.tyFB.tyBtnEnt.uiMaskRtStat));
			fUIInRtStatOff(ADR(tyP0933PullConv.tyFB.tyBtnExit.uiMaskRtStat));
			fUIInRtStatOff(ADR(tyP0933PullConv.tyFB.tyBtnExt.uiMaskRtStat));
			fUIInRtStatOff(ADR(tyP0933PullConv.tyFB.tyBtnRet.uiMaskRtStat));
			fUIInRtStatHide(ADR(tyP0933PullConv.tyFB.tyBtnRotToHm.uiMaskRtStat));
			fUIInRtStatHide(ADR(tyP0933PullConv.tyFB.tyBtnRotToRm.uiMaskRtStat));
			fUIInRtStatOff(ADR(tyP0933PullConv.tyCom.tyBtnSwitch.uiMaskRtStat));

		ELSE

			fUIInRtStatHide(ADR(tyP0933PullConv.tyFB.tyBtnCylEnt.uiMaskRtStat));
			fUIInRtStatHide(ADR(tyP0933PullConv.tyFB.tyBtnEnt.uiMaskRtStat));
			fUIInRtStatHide(ADR(tyP0933PullConv.tyFB.tyBtnExit.uiMaskRtStat));
			fUIInRtStatHide(ADR(tyP0933PullConv.tyFB.tyBtnExt.uiMaskRtStat));
			fUIInRtStatHide(ADR(tyP0933PullConv.tyFB.tyBtnRet.uiMaskRtStat));
			fUIInRtStatHide(ADR(tyP0933PullConv.tyFB.tyBtnRotToHm.uiMaskRtStat));
			fUIInRtStatHide(ADR(tyP0933PullConv.tyFB.tyBtnRotToRm.uiMaskRtStat));
			fUIInRtStatHide(ADR(tyP0933PullConv.tyCom.tyBtnSwitch.uiMaskRtStat));

		END_IF
	END_IF

	IF p_bLifterBtmSltAPosDiff OR (p_bTravAPosDiff AND p_bTravBPosDiff AND p_bTravCPosDiff)
		OR p_tyDI.bInShutterOpenRS = FALSE
		THEN
		//	fUIInRtStatOff(ADR(tyP0933PullConv.tyFB.tyBtnCylEnt.uiMaskRtStat));
		//	fUIInRtStatOff(ADR(tyP0933PullConv.tyFB.tyBtnEnt.uiMaskRtStat));
			fUIInRtStatOff(ADR(tyP0933PullConv.tyFB.tyBtnExt.uiMaskRtStat));
	END_IF

	IF p_tyDI.bPullerExtRS = FALSE THEN
		fUIInRtStatOff(ADR(tyP0933PullConv.tyFB.tyBtnRotToRm.uiMaskRtStat));
	ELSE
		fUIInRtStatHide(ADR(tyP0933PullConv.tyFB.tyBtnRotToRm.uiMaskRtStat));
	END_IF

	//Shutter Control
	IF tyP0933PullConv.tyInOutletShutterFB.tyBtnOpen.bRtCompl = TRUE THEN
		tyP0933PullConv.tyInOutletShutterFB.tyBtnOpen.bRtCompl	:= FALSE;

		tyP0933PullConv.tyInOutletShutterFB.tyBtnOpen.bValue	:= TRUE;
		tyP0933PullConv.tyInOutletShutterFB.tyBtnClose.bValue	:= FALSE;

	ELSIF tyP0933PullConv.tyInOutletShutterFB.tyBtnClose.bRtCompl = TRUE THEN
		tyP0933PullConv.tyInOutletShutterFB.tyBtnClose.bRtCompl	:= FALSE;

		tyP0933PullConv.tyInOutletShutterFB.tyBtnClose.bValue	:= TRUE;
		tyP0933PullConv.tyInOutletShutterFB.tyBtnOpen.bValue	:= FALSE;
	END_IF

	IF tyP0933PullConv.tyInOutletShutterFB.tyBtnOpen.bValue = TRUE THEN
		eInShutterAct	:= PneuActRet;
		eOutShutterAct	:= PneuActRet;

		IF (p_eInShutterStat = PneuActRet AND p_eInShutterStatus = Done)
			AND (p_eOutShutterStat = PneuActRet AND p_eOutShutterStatus = Done)
			THEN
			eInShutterAct	:= PneuActIdle;
			eOutShutterAct	:= PneuActIdle;
			tyP0933PullConv.tyInOutletShutterFB.tyBtnOpen.bValue	:= FALSE;
		ELSIF p_eInShutterStatus = Error OR p_eOutShutterStatus = Error THEN
			tyP0933PullConv.tyInOutletShutterFB.tyBtnOpen.bValue	:= FALSE;
		END_IF

	ELSIF tyP0933PullConv.tyInOutletShutterFB.tyBtnClose.bValue = TRUE THEN
		eInShutterAct	:= PneuActExt;
		eOutShutterAct	:= PneuActExt;
		IF (p_eInShutterStat = PneuActExt AND p_eInShutterStatus = Done)
			AND (p_eOutShutterStat = PneuActExt AND p_eOutShutterStatus = Done)
			THEN
			eInShutterAct	:= PneuActIdle;
			eOutShutterAct	:= PneuActIdle;
			tyP0933PullConv.tyInOutletShutterFB.tyBtnClose.bValue := FALSE;
		ELSIF p_eInShutterStatus = Error OR p_eOutShutterStatus = Error THEN
			tyP0933PullConv.tyInOutletShutterFB.tyBtnClose.bValue := FALSE;
		END_IF
	END_IF

	tyP0933PullConv.tyFB.tyBtnRet.uiMaskRtStat	:= TRUE;
	tyP0933PullConv.tyFB.tyBtnExt.uiMaskRtStat	:= TRUE;

END_ACTION
```

#### Act_OptP0933PullerConvFBStat.st
```iecst
ACTION Act_OptP0933PullerConvFBStat:

//	IF p_tyNtParamCurr.bProjPullerRotCylPrep = FALSE AND p_tyNtParamCurr.bProjMotorizedPullerPrep = FALSE THEN
//		tyP0933PullConv.tyFB.tyStringStat.sValue   := p_sPullConvStatTxt;
//	ELSIF p_tyNtParamCurr.bProjPullerRotCylPrep = TRUE AND p_tyNtParamCurr.bProjMotorizedPullerPrep = FALSE THEN
//		IF tyP0933PullConv.tyFB.tyBtnExt.bRtCompl OR tyP0933PullConv.tyFB.tyBtnRet.bRtCompl THEN
//			tyP0933PullConv.tyFB.tyStringStat.sValue   := p_sPullerStatTxt;
//		ELSE
//			tyP0933PullConv.tyFB.tyStringStat.sValue   := p_sPullConvStatTxt;
//		END_IF
//	ELSIF p_tyNtParamCurr.bProjPullerRotCylPrep = TRUE AND p_tyNtParamCurr.bProjMotorizedPullerPrep = TRUE THEN
//		IF tyP0933PullConv.tyFB.tyBtnExt.bRtCompl OR tyP0933PullConv.tyFB.tyBtnRet.bRtCompl THEN
//			tyP0933PullConv.tyFB.tyStringStat.sValue   := p_sMtrPshrStatTxt;
//		ELSE
//			tyP0933PullConv.tyFB.tyStringStat.sValue   := p_sPullConvStatTxt;
//		END_IF
//	END_IF

	tyP0933PullConv.tyFB.tyStringStat.sValue   := p_sPullConvStatTxt;

END_ACTION
```

#### Act_OptP0933PullerConvDC.st
```iecst
ACTION Act_OptP0933PullerConvDC:

	//Conveyor
	IF tyP0933PullConv.tyDC.tyBtnStop.bRtCompl = TRUE THEN
		ePullConvAct	:= ConvActStop;

		IF p_ePullConvStat = ConvActStop AND p_ePullConvStatus = Done THEN
			ePullConvAct	:= ConvActIdle;

			tyP0933PullConv.tyDC.tyBtnStop.bRtCompl		:= FALSE;
			tyP0933PullConv.tyDC.tyBtnStop.bValue		:= TRUE;
			tyP0933PullConv.tyDC.tyBtnStop.bRtLk		:= TRUE;

			tyP0933PullConv.tyDC.tyBtnStart.bRtCompl	:= FALSE;
			tyP0933PullConv.tyDC.tyBtnStart.bValue		:= FALSE;
			tyP0933PullConv.tyDC.tyBtnStart.bRtLk		:= FALSE;
		END_IF

	ELSIF tyP0933PullConv.tyDC.tyBtnStart.bRtCompl = TRUE THEN
		tyP0933PullConv.tyDC.tyBtnStart.bValue	:= TRUE;
		tyP0933PullConv.tyDC.tyBtnStart.bRtLk	:= TRUE;

		tyP0933PullConv.tyDC.tyBtnStop.bValue	:= FALSE;
		tyP0933PullConv.tyDC.tyBtnStop.bRtLk	:= FALSE;

		ePullConvAct	:= ConvActSetMtrSigOnOrLToR;

		IF p_ePullConvStat = ConvActSetMtrSigOnOrLToR AND p_ePullConvStatus = Done THEN
			ePullConvAct	:= ConvActIdle;

			tyP0933PullConv.tyDC.tyBtnStart.bRtCompl	:= FALSE;
		END_IF

	END_IF

	//Puller
	IF p_tyNtParamCurr.bProjPullerRotCylPrep = TRUE THEN

		IF tyP0933PullConv.tyCom.tyBtnSwitch.bValue = TRUE THEN

			IF p_bPullConvPullerTwoOutputCtrl = FALSE THEN

				IF tyP0933PullConv.tyDC.tyBtnRet.bRtCompl = TRUE THEN
					tyP0933PullConv.tyDC.tyBtnRet.bValue	:= TRUE;
					tyP0933PullConv.tyDC.tyBtnExt.bValue	:= FALSE;

					ePullConvAct	:= ConvActPullerSetRet;

					IF p_ePullConvStat = ConvActPullerSetRet AND p_ePullConvStatus = Done THEN
						ePullConvAct	:= ConvActIdle;

						tyP0933PullConv.tyDC.tyBtnRet.bRtCompl	:= FALSE;
					END_IF

				ELSIF tyP0933PullConv.tyDC.tyBtnExt.bRtCompl = TRUE THEN
					tyP0933PullConv.tyDC.tyBtnExt.bValue	:= TRUE;
					tyP0933PullConv.tyDC.tyBtnRet.bValue	:= FALSE;

					ePullConvAct	:= ConvActPullerSetExt;

					IF p_ePullConvStat = ConvActPullerSetExt AND p_ePullConvStatus = Done THEN
						ePullConvAct	:= ConvActIdle;

						tyP0933PullConv.tyDC.tyBtnExt.bRtCompl	:= FALSE;
					END_IF

				END_IF

			ELSE

				IF (tyP0933PullConv.tyDC.tyBtnRet.bRtCompl = TRUE) OR (tyP0933PullConv.tyDC.tyBtnExt.bRtCompl = TRUE) THEN
					IF (tyP0933PullConv.tyDC.tyBtnRet.bValue = TRUE) AND (tyP0933PullConv.tyDC.tyBtnExt.bValue = TRUE) THEN
						ePullConvAct	:= ConvActPullerSetAll;

						IF p_ePullConvStat = ConvActPullerSetAll AND p_ePullConvStatus = Done THEN
							ePullConvAct	:= ConvActIdle;

							tyP0933PullConv.tyDC.tyBtnRet.bRtCompl	:= FALSE;
							tyP0933PullConv.tyDC.tyBtnExt.bRtCompl	:= FALSE;
						END_IF

					ELSIF (tyP0933PullConv.tyDC.tyBtnRet.bValue = TRUE) AND (tyP0933PullConv.tyDC.tyBtnExt.bValue = FALSE) THEN
						ePullConvAct	:= ConvActPullerSetRet;

						IF p_ePullConvStat = ConvActPullerSetRet AND p_ePullConvStatus = Done THEN
							ePullConvAct	:= ConvActIdle;

							tyP0933PullConv.tyDC.tyBtnRet.bRtCompl	:= FALSE;
							tyP0933PullConv.tyDC.tyBtnExt.bRtCompl	:= FALSE;
						END_IF

					ELSIF (tyP0933PullConv.tyDC.tyBtnRet.bValue = FALSE) AND (tyP0933PullConv.tyDC.tyBtnExt.bValue = TRUE) THEN
						ePullConvAct	:= ConvActPullerSetExt;

						IF p_ePullConvStat = ConvActPullerSetExt AND p_ePullConvStatus = Done THEN
							ePullConvAct	:= ConvActIdle;

							tyP0933PullConv.tyDC.tyBtnRet.bRtCompl	:= FALSE;
							tyP0933PullConv.tyDC.tyBtnExt.bRtCompl	:= FALSE;
						END_IF

					ELSE
						ePullConvAct	:= ConvActPullerRstAll;

						IF p_ePullConvStat = ConvActPullerRstAll AND p_ePullConvStatus = Done THEN
							ePullConvAct	:= ConvActIdle;

							tyP0933PullConv.tyDC.tyBtnRet.bRtCompl	:= FALSE;
							tyP0933PullConv.tyDC.tyBtnExt.bRtCompl	:= FALSE;
						END_IF

					END_IF

				END_IF

			END_IF

			tyP0933PullConv.tyFB.tyBtnExt.bRtCompl	:= FALSE;
			tyP0933PullConv.tyFB.tyBtnExt.bValue	:= FALSE;
			tyP0933PullConv.tyFB.tyBtnRet.bRtCompl	:= FALSE;
			tyP0933PullConv.tyFB.tyBtnRet.bValue	:= FALSE;

		END_IF

	ELSE

		IF tyP0933PullConv.tyCom.tyBtnSwitch.bValue = TRUE THEN

			IF p_bPullerTwoCtrlOut = FALSE THEN

				IF tyP0933PullConv.tyDC.tyBtnRet.bRtCompl = TRUE THEN
					tyP0933PullConv.tyDC.tyBtnRet.bValue	:= TRUE;
					tyP0933PullConv.tyDC.tyBtnExt.bValue	:= FALSE;

					ePullerAct	:= PneuActSetRet;

					IF p_ePullerStat = PneuActSetRet AND p_ePullerStatus = Done THEN
						ePullerAct	:= PneuActIdle;

						tyP0933PullConv.tyDC.tyBtnRet.bRtCompl	:= FALSE;
					END_IF

				ELSIF tyP0933PullConv.tyDC.tyBtnExt.bRtCompl = TRUE THEN
					tyP0933PullConv.tyDC.tyBtnExt.bValue	:= TRUE;
					tyP0933PullConv.tyDC.tyBtnRet.bValue	:= FALSE;

					ePullerAct	:= PneuActSetExt;

					IF p_ePullerStat = PneuActSetExt AND p_ePullerStatus = Done THEN
						ePullerAct	:= PneuActIdle;

						tyP0933PullConv.tyDC.tyBtnExt.bRtCompl	:= FALSE;
					END_IF

				END_IF

			ELSE

				IF (tyP0933PullConv.tyDC.tyBtnRet.bRtCompl = TRUE) OR (tyP0933PullConv.tyDC.tyBtnExt.bRtCompl = TRUE) THEN
					IF (tyP0933PullConv.tyDC.tyBtnRet.bValue = TRUE) AND (tyP0933PullConv.tyDC.tyBtnExt.bValue = TRUE) THEN

						ePullerAct	:= PneuActSetAll;

						IF p_ePullerStat = PneuActSetAll AND p_ePullerStatus = Done THEN
							ePullerAct	:= PneuActIdle;

							tyP0933PullConv.tyDC.tyBtnRet.bRtCompl	:= FALSE;
							tyP0933PullConv.tyDC.tyBtnExt.bRtCompl	:= FALSE;
						END_IF

					ELSIF (tyP0933PullConv.tyDC.tyBtnRet.bValue = TRUE) AND (tyP0933PullConv.tyDC.tyBtnExt.bValue = FALSE) THEN

						ePullerAct	:= PneuActSetRet;

						IF p_ePullerStat = PneuActSetRet AND p_ePullerStatus = Done THEN
							ePullerAct	:= PneuActIdle;

							tyP0933PullConv.tyDC.tyBtnRet.bRtCompl	:= FALSE;
							tyP0933PullConv.tyDC.tyBtnExt.bRtCompl	:= FALSE;
						END_IF

					ELSIF (tyP0933PullConv.tyDC.tyBtnRet.bValue = FALSE) AND (tyP0933PullConv.tyDC.tyBtnExt.bValue = TRUE) THEN

						ePullerAct	:= PneuActSetExt;

						IF p_ePullerStat = PneuActSetExt AND p_ePullerStatus = Done THEN
							ePullerAct	:= PneuActIdle;

							tyP0933PullConv.tyDC.tyBtnRet.bRtCompl	:= FALSE;
							tyP0933PullConv.tyDC.tyBtnExt.bRtCompl	:= FALSE;
						END_IF

					ELSE

						ePullerAct	:= PneuActRstAll;

						IF p_ePullerStat = PneuActRstAll AND p_ePullerStatus = Done THEN
							ePullerAct	:= PneuActIdle;

							tyP0933PullConv.tyDC.tyBtnRet.bRtCompl	:= FALSE;
							tyP0933PullConv.tyDC.tyBtnExt.bRtCompl	:= FALSE;
						END_IF

					END_IF

				END_IF

			END_IF

			tyP0933PullConv.tyFB.tyBtnExt.bRtCompl	:= FALSE;
			tyP0933PullConv.tyFB.tyBtnExt.bValue	:= FALSE;
			tyP0933PullConv.tyFB.tyBtnRet.bRtCompl	:= FALSE;
			tyP0933PullConv.tyFB.tyBtnRet.bValue	:= FALSE;

		END_IF

	END_IF

	//Rotating Cylinder
	IF tyP0933PullConv.tyCom.tyBtnSwitch.bValue = TRUE THEN

		IF p_bPullConvRotTwoOutputCtrl = FALSE THEN

			IF tyP0933PullConv.tyDC.tyBtnRotToHm.bRtCompl = TRUE THEN
				tyP0933PullConv.tyDC.tyBtnRotToHm.bValue	:= TRUE;
				tyP0933PullConv.tyDC.tyBtnRotToRm.bValue	:= FALSE;

				ePullConvAct	:= ConvActRotSetHome;

				IF p_ePullConvStat = ConvActRotSetHome AND p_ePullConvStatus = Done THEN
					ePullConvAct	:= ConvActIdle;

					tyP0933PullConv.tyDC.tyBtnRotToHm.bRtCompl	:= FALSE;
				END_IF

			ELSIF tyP0933PullConv.tyDC.tyBtnRotToRm.bRtCompl = TRUE THEN
				tyP0933PullConv.tyDC.tyBtnRotToRm.bValue	:= TRUE;
				tyP0933PullConv.tyDC.tyBtnRotToHm.bValue	:= FALSE;

				ePullConvAct	:= ConvActRotSetRmt;

				IF p_ePullConvStat = ConvActRotSetRmt AND p_ePullConvStatus = Done THEN
					ePullConvAct	:= ConvActIdle;

					tyP0933PullConv.tyDC.tyBtnRotToRm.bRtCompl	:= FALSE;
				END_IF

			END_IF

		ELSE

			IF (tyP0933PullConv.tyDC.tyBtnRotToHm.bRtCompl = TRUE) OR (tyP0933PullConv.tyDC.tyBtnRotToRm.bRtCompl = TRUE) THEN
				IF (tyP0933PullConv.tyDC.tyBtnRotToHm.bValue = TRUE) AND (tyP0933PullConv.tyDC.tyBtnRotToRm.bValue = TRUE) THEN
					ePullConvAct	:= ConvActRotSetAll;

					IF p_ePullConvStat = ConvActRotSetAll AND p_ePullConvStatus = Done THEN
						ePullConvAct	:= ConvActIdle;

						tyP0933PullConv.tyDC.tyBtnRotToHm.bRtCompl	:= FALSE;
						tyP0933PullConv.tyDC.tyBtnRotToRm.bRtCompl	:= FALSE;
					END_IF

				ELSIF (tyP0933PullConv.tyDC.tyBtnRotToHm.bValue = TRUE) AND (tyP0933PullConv.tyDC.tyBtnRotToRm.bValue = FALSE) THEN
					ePullConvAct	:= ConvActRotSetHome;

					IF p_ePullConvStat = ConvActRotSetHome AND p_ePullConvStatus = Done THEN
						ePullConvAct	:= ConvActIdle;

						tyP0933PullConv.tyDC.tyBtnRotToHm.bRtCompl	:= FALSE;
						tyP0933PullConv.tyDC.tyBtnRotToRm.bRtCompl	:= FALSE;
					END_IF

				ELSIF (tyP0933PullConv.tyDC.tyBtnRotToHm.bValue = FALSE) AND (tyP0933PullConv.tyDC.tyBtnRotToRm.bValue = TRUE) THEN
					ePullConvAct	:= ConvActRotSetRmt;

					IF p_ePullConvStat = ConvActRotSetRmt AND p_ePullConvStatus = Done THEN
						ePullConvAct	:= ConvActIdle;

						tyP0933PullConv.tyDC.tyBtnRotToHm.bRtCompl	:= FALSE;
						tyP0933PullConv.tyDC.tyBtnRotToRm.bRtCompl	:= FALSE;
					END_IF

				ELSE
					ePullConvAct	:= ConvActRotRstAll;

					IF p_ePullConvStat = ConvActRotRstAll AND p_ePullConvStatus = Done THEN
						ePullConvAct	:= ConvActIdle;

						tyP0933PullConv.tyDC.tyBtnRotToHm.bRtCompl	:= FALSE;
						tyP0933PullConv.tyDC.tyBtnRotToRm.bRtCompl	:= FALSE;
					END_IF

				END_IF

			END_IF

		END_IF

		tyP0933PullConv.tyFB.tyBtnRotToRm.bRtCompl	:= FALSE;
		tyP0933PullConv.tyFB.tyBtnRotToRm.bValue	:= FALSE;
		tyP0933PullConv.tyFB.tyBtnRotToHm.bRtCompl	:= FALSE;
		tyP0933PullConv.tyFB.tyBtnRotToHm.bValue	:= FALSE;

	END_IF

	//For Motorized Puller
	IF tyP0933PullConv.tyDC.tyBtnAlarmRst.bRtCompl = TRUE THEN

		IF tyP0933PullConv.tyDC.tyBtnAlarmRst.bValue = TRUE THEN
			eMtrPshrAct	:= MtrPshrActSetAlmRst;

			IF p_eMtrPshrStat = MtrPshrActSetAlmRst AND p_eMtrPshrStatus = Done THEN
				eMtrPshrAct	:= MtrPshrActIdle;

				tyP0933PullConv.tyDC.tyBtnAlarmRst.bRtCompl	:= FALSE;
			END_IF
		ELSE
			eMtrPshrAct	:= MtrPshrActRstAlmRst;

			IF p_eMtrPshrStat = MtrPshrActRstAlmRst AND p_eMtrPshrStatus = Done THEN
				eMtrPshrAct	:= MtrPshrActIdle;

				tyP0933PullConv.tyDC.tyBtnAlarmRst.bRtCompl	:= FALSE;
			END_IF
		END_IF

	ELSIF tyP0933PullConv.tyDC.tyBtnBrake.bRtCompl = TRUE THEN

		IF tyP0933PullConv.tyDC.tyBtnBrake.bValue = TRUE THEN
			eMtrPshrAct	:= MtrPshrActSetBrake;

			IF p_eMtrPshrStat = MtrPshrActSetBrake AND p_eMtrPshrStatus = Done THEN
				eMtrPshrAct	:= MtrPshrActIdle;

				tyP0933PullConv.tyDC.tyBtnBrake.bRtCompl	:= FALSE;
			END_IF
		ELSE
			eMtrPshrAct	:= MtrPshrActRstBrake;

			IF p_eMtrPshrStat = MtrPshrActRstBrake AND p_eMtrPshrStatus = Done THEN
				eMtrPshrAct	:= MtrPshrActIdle;

				tyP0933PullConv.tyDC.tyBtnBrake.bRtCompl	:= FALSE;
			END_IF
		END_IF

	ELSIF tyP0933PullConv.tyDC.tyBtnSigOn.bRtCompl = TRUE THEN

		IF tyP0933PullConv.tyDC.tyBtnSigOn.bValue = TRUE THEN
			eMtrPshrAct	:= MtrPshrActSetSigOn;

			IF p_eMtrPshrStat = MtrPshrActSetSigOn AND p_eMtrPshrStatus = Done THEN
				eMtrPshrAct	:= MtrPshrActIdle;

				tyP0933PullConv.tyDC.tyBtnSigOn.bRtCompl	:= FALSE;
			END_IF
		ELSE
			eMtrPshrAct	:= MtrPshrActRstSigOn;

			IF p_eMtrPshrStat = MtrPshrActRstSigOn AND p_eMtrPshrStatus = Done THEN
				eMtrPshrAct	:= MtrPshrActIdle;

				tyP0933PullConv.tyDC.tyBtnSigOn.bRtCompl	:= FALSE;
			END_IF
		END_IF

	ELSIF tyP0933PullConv.tyDC.tyBtnSpdBinBit0.bRtCompl = TRUE THEN

		IF tyP0933PullConv.tyDC.tyBtnSpdBinBit0.bValue = TRUE THEN
			eMtrPshrAct	:= MtrPshrActSetSpdBit0;

			IF p_eMtrPshrStat = MtrPshrActSetSpdBit0 AND p_eMtrPshrStatus = Done THEN
				eMtrPshrAct	:= MtrPshrActIdle;

				tyP0933PullConv.tyDC.tyBtnSpdBinBit0.bRtCompl	:= FALSE;
			END_IF
		ELSE
			eMtrPshrAct	:= MtrPshrActRstSpdBit0;

			IF p_eMtrPshrStat = MtrPshrActRstSpdBit0 AND p_eMtrPshrStatus = Done THEN
				eMtrPshrAct	:= MtrPshrActIdle;

				tyP0933PullConv.tyDC.tyBtnSpdBinBit0.bRtCompl	:= FALSE;
			END_IF
		END_IF

	ELSIF tyP0933PullConv.tyDC.tyBtnSpdBinBit1.bRtCompl = TRUE THEN

		IF tyP0933PullConv.tyDC.tyBtnSpdBinBit1.bValue = TRUE THEN
			eMtrPshrAct	:= MtrPshrActSetSpdBit1;

			IF p_eMtrPshrStat = MtrPshrActSetSpdBit1 AND p_eMtrPshrStatus = Done THEN
				eMtrPshrAct	:= MtrPshrActIdle;

				tyP0933PullConv.tyDC.tyBtnSpdBinBit1.bRtCompl	:= FALSE;
			END_IF
		ELSE
			eMtrPshrAct	:= MtrPshrActRstSpdBit1;

			IF p_eMtrPshrStat = MtrPshrActRstSpdBit1 AND p_eMtrPshrStatus = Done THEN
				eMtrPshrAct	:= MtrPshrActIdle;

				tyP0933PullConv.tyDC.tyBtnSpdBinBit1.bRtCompl	:= FALSE;
			END_IF
		END_IF

	ELSIF tyP0933PullConv.tyDC.tyBtnSpdBinBit2.bRtCompl = TRUE THEN

		IF tyP0933PullConv.tyDC.tyBtnSpdBinBit2.bValue = TRUE THEN
			eMtrPshrAct	:= MtrPshrActSetSpdBit2;

			IF p_eMtrPshrStat = MtrPshrActSetSpdBit2 AND p_eMtrPshrStatus = Done THEN
				eMtrPshrAct	:= MtrPshrActIdle;

				tyP0933PullConv.tyDC.tyBtnSpdBinBit2.bRtCompl	:= FALSE;
			END_IF
		ELSE
			eMtrPshrAct	:= MtrPshrActRstSpdBit2;

			IF p_eMtrPshrStat = MtrPshrActRstSpdBit2 AND p_eMtrPshrStatus = Done THEN
				eMtrPshrAct	:= MtrPshrActIdle;

				tyP0933PullConv.tyDC.tyBtnSpdBinBit2.bRtCompl	:= FALSE;
			END_IF
		END_IF

	END_IF

	//Mask
	IF p_ePullConvStatus = Error OR p_ePullerStatus = Error THEN

		fUIInRtStatOff(ADR(tyP0933PullConv.tyDC.tyBtnStart.uiMaskRtStat));
		fUIInRtStatOff(ADR(tyP0933PullConv.tyDC.tyBtnExt.uiMaskRtStat));
		fUIInRtStatOff(ADR(tyP0933PullConv.tyDC.tyBtnRet.uiMaskRtStat));
		fUIInRtStatOff(ADR(tyP0933PullConv.tyDC.tyBtnRotToHm.uiMaskRtStat));
		fUIInRtStatOff(ADR(tyP0933PullConv.tyDC.tyBtnRotToRm.uiMaskRtStat));

	ELSIF tyP0933PullConv.tyDC.tyBtnStart.bValue = TRUE THEN

		fUIInRtStatHide(ADR(tyP0933PullConv.tyDC.tyBtnStart.uiMaskRtStat));
		fUIInRtStatOff(ADR(tyP0933PullConv.tyDC.tyBtnExt.uiMaskRtStat));
		fUIInRtStatOff(ADR(tyP0933PullConv.tyDC.tyBtnRet.uiMaskRtStat));
		fUIInRtStatOff(ADR(tyP0933PullConv.tyDC.tyBtnRotToHm.uiMaskRtStat));
		fUIInRtStatOff(ADR(tyP0933PullConv.tyDC.tyBtnRotToRm.uiMaskRtStat));

	ELSE

		fUIInRtStatHide(ADR(tyP0933PullConv.tyDC.tyBtnStart.uiMaskRtStat));
		fUIInRtStatHide(ADR(tyP0933PullConv.tyDC.tyBtnExt.uiMaskRtStat));
		fUIInRtStatHide(ADR(tyP0933PullConv.tyDC.tyBtnRet.uiMaskRtStat));
		fUIInRtStatHide(ADR(tyP0933PullConv.tyDC.tyBtnRotToHm.uiMaskRtStat));
		fUIInRtStatHide(ADR(tyP0933PullConv.tyDC.tyBtnRotToRm.uiMaskRtStat));

	END_IF

	//Mask
//	tyP0933PullConv.tyDC.tyBtnExt.uiMaskRtStat.0		:= NOT(p_eMtrPshrStatus = Error OR tyP0933PullConv.tyDC.tyBtnRet.bValue);
	tyP0933PullConv.tyDC.tyBtnRet.uiMaskRtStat.0		:= NOT(p_eMtrPshrStatus = Error OR tyP0933PullConv.tyDC.tyBtnExt.bValue);
	tyP0933PullConv.tyDC.tyBtnSigOn.uiMaskRtStat.0		:= NOT(p_eMtrPshrStatus = Error);
	tyP0933PullConv.tyDC.tyBtnAlarmRst.uiMaskRtStat.0	:= NOT(p_eMtrPshrStatus = Error);
	tyP0933PullConv.tyDC.tyBtnBrake.uiMaskRtStat.0		:= NOT(p_eMtrPshrStatus = Error);
	tyP0933PullConv.tyDC.tyBtnSpdBinBit0.uiMaskRtStat.0	:= NOT(p_eMtrPshrStatus = Error);
	tyP0933PullConv.tyDC.tyBtnSpdBinBit1.uiMaskRtStat.0	:= NOT(p_eMtrPshrStatus = Error);
	tyP0933PullConv.tyDC.tyBtnSpdBinBit2.uiMaskRtStat.0	:= NOT(p_eMtrPshrStatus = Error);

	IF p_bLifterBtmSltAPosDiff OR (p_bTravAPosDiff AND p_bTravBPosDiff AND p_bTravCPosDiff)
		OR p_eMtrPshrStatus = Error
		THEN
		fUIInRtStatOff(ADR(tyP0933PullConv.tyDC.tyBtnExt.uiMaskRtStat));
	END_IF

END_ACTION
```

#### Act_OptP0933PullerConvRstMnl.st
```iecst
ACTION Act_OptP0933RstMnl:

	IF EDGEPOS((bManualMod = FALSE) OR (p_ePullConvStatus = Error OR p_ePullerStatus = Error)) THEN

		ePullConvAct	:= ConvActIdle;
		ePullerAct		:= PneuActIdle;

		//FB - Motor
		tyP0933PullConv.tyFB.tyBtnCylEnt.bRtCompl				:= FALSE;
		tyP0933PullConv.tyFB.tyBtnEnt.bRtCompl					:= FALSE;
		tyP0933PullConv.tyFB.tyBtnExit.bRtCompl					:= FALSE;
		tyP0933PullConv.tyFB.tyBtnStop.bRtCompl					:= FALSE;

		tyP0933PullConv.tyFB.tyBtnCylEnt.bValue					:= FALSE;
		tyP0933PullConv.tyFB.tyBtnEnt.bValue					:= FALSE;
		tyP0933PullConv.tyFB.tyBtnExit.bValue					:= FALSE;
		tyP0933PullConv.tyFB.tyBtnStop.bValue					:= TRUE;

		tyP0933PullConv.tyFB.tyBtnCylEnt.bRtLk					:= FALSE;
		tyP0933PullConv.tyFB.tyBtnEnt.bRtLk						:= FALSE;
		tyP0933PullConv.tyFB.tyBtnExit.bRtLk					:= FALSE;
		tyP0933PullConv.tyFB.tyBtnStop.bRtLk					:= TRUE;

		tyP0933PullConv.tyFB.tyBtnCylEnt.uiMaskRtStat.0			:= TRUE;
		tyP0933PullConv.tyFB.tyBtnEnt.uiMaskRtStat.0			:= TRUE;
		tyP0933PullConv.tyFB.tyBtnExit.uiMaskRtStat.0			:= TRUE;
		tyP0933PullConv.tyCom.tyBtnSwitch.uiMaskRtStat.0		:= TRUE;

		//FB - Pneu
		tyP0933PullConv.tyFB.tyBtnExt.bRtCompl					:= FALSE;
		tyP0933PullConv.tyFB.tyBtnRet.bRtCompl					:= FALSE;
		tyP0933PullConv.tyFB.tyBtnRotToHm.bRtCompl				:= FALSE;
		tyP0933PullConv.tyFB.tyBtnRotToRm.bRtCompl				:= FALSE;

		tyP0933PullConv.tyFB.tyBtnExt.bValue					:= FALSE;
		tyP0933PullConv.tyFB.tyBtnRet.bValue					:= FALSE;
		tyP0933PullConv.tyFB.tyBtnRotToHm.bValue				:= FALSE;
		tyP0933PullConv.tyFB.tyBtnRotToRm.bValue				:= FALSE;

		tyP0933PullConv.tyFB.tyBtnExt.uiMaskRtStat.0			:= TRUE;
		tyP0933PullConv.tyFB.tyBtnRet.uiMaskRtStat.0			:= TRUE;
		tyP0933PullConv.tyFB.tyBtnRotToHm.uiMaskRtStat.0		:= TRUE;
		tyP0933PullConv.tyFB.tyBtnRotToRm.uiMaskRtStat.0		:= TRUE;

		//DC - Motor
		tyP0933PullConv.tyDC.tyBtnStart.bRtCompl				:= FALSE;
		tyP0933PullConv.tyDC.tyBtnStop.bRtCompl					:= FALSE;

		tyP0933PullConv.tyDC.tyBtnStart.bValue					:= FALSE;
		tyP0933PullConv.tyDC.tyBtnStop.bValue					:= TRUE;

		tyP0933PullConv.tyDC.tyBtnStart.bRtLk					:= FALSE;
		tyP0933PullConv.tyDC.tyBtnStop.bRtLk					:= TRUE;

		tyP0933PullConv.tyDC.tyBtnStart.uiMaskRtStat.0			:= TRUE;
		tyP0933PullConv.tyCom.tyBtnSwitch.uiMaskRtStat.0		:= TRUE;

		//DC - Pneu
		tyP0933PullConv.tyDC.tyBtnExt.bRtCompl					:= FALSE;
		tyP0933PullConv.tyDC.tyBtnRet.bRtCompl					:= FALSE;
		tyP0933PullConv.tyDC.tyBtnRotToHm.bRtCompl				:= FALSE;
		tyP0933PullConv.tyDC.tyBtnRotToRm.bRtCompl				:= FALSE;

		tyP0933PullConv.tyDC.tyBtnExt.bValue					:= FALSE;
		tyP0933PullConv.tyDC.tyBtnRet.bValue					:= FALSE;
		tyP0933PullConv.tyDC.tyBtnRotToHm.bValue				:= FALSE;
		tyP0933PullConv.tyDC.tyBtnRotToRm.bValue				:= FALSE;

		tyP0933PullConv.tyDC.tyBtnExt.uiMaskRtStat.0			:= TRUE;
		tyP0933PullConv.tyDC.tyBtnRet.uiMaskRtStat.0			:= TRUE;
		tyP0933PullConv.tyDC.tyBtnRotToHm.uiMaskRtStat.0		:= TRUE;
		tyP0933PullConv.tyDC.tyBtnRotToRm.uiMaskRtStat.0		:= TRUE;

	END_IF

	IF EDGEPOS(bManualMod = FALSE) THEN
		tyP0933PullConv.tyCom.tyBtnSwitch.bValue := FALSE;

		fUIInRtStatHide(ADR(tyP0933PullConv.tyDC.tyLyr.uiRtStat));
		fUIInRtStatOff(ADR(tyP0933PullConv.tyFB.tyLyr.uiRtStat));

	END_IF

	eInShutterAct	:= PneuActIdle;
	eOutShutterAct	:= PneuActIdle;

	tyP0933PullConv.tyInOutletShutterFB.tyBtnClose.bRtCompl	:= FALSE;
	tyP0933PullConv.tyInOutletShutterFB.tyBtnClose.bValue	:= FALSE;
	tyP0933PullConv.tyInOutletShutterFB.tyBtnOpen.bRtCompl	:= FALSE;
	tyP0933PullConv.tyInOutletShutterFB.tyBtnOpen.bValue	:= FALSE;

END_ACTION
```

#### Act_EntP0934Disp.st
```iecst
ACTION Act_EntP0934Disp:

	//Access Address
	p_tyC0001MotionStd ACCESS ADR(tyP0934AW.tyMotionStd);

	p_tyC0002FullMask ACCESS ADR(tyP0934AW.tyFullMaskHide);

	p_tyC0004Navi ACCESS ADR(tyP0934AW.tyNaviBack);

	p_tyC0005Main ACCESS ADR(tyCommon.tyMain);

	p_tyC0007Notif ACCESS ADR(tyCommon.tyNotif);

	p_tyC0008MsgBox ACCESS ADR(tyP0934AW.tyMsgBoxHide);

	p_tyC0009Info ACCESS ADR(tyCommon.tyInfo);

	p_tyP0934AW ACCESS ADR(tyP0934AW.tyAW);

	//Display
	tyP0934AW.tyAW.tyNumNewWidth.diValue	:= p_tyProdRcpCurrRcp0.diWidthInUM;

	tyP0934AW.tyMotionStd.tyBtnPwr.bValue	:= p_bAWOpenPwrOn;

END_ACTION
```

#### Act_OptP0934FBCtrl.st
```iecst
ACTION Act_OptP0934FBCtrl:

	fbJogSlowToFastDlyTm.PT	:= T#2s;
	fbJogSlowToFastDlyTm;
	fbLmtRstTm;

	//Conveyor Sensor Interruption
	IF (p_tyDI.bConvLftSen OR p_tyDI.bConvRgtSen OR p_tyDI.bPullerRetRS = FALSE) AND eCurrPage = UIP0934AW THEN
		tyP0934AW.tyMotionStd.tyBtnStop.bRtCompl	:= TRUE;
	END_IF

//	IF EDGEPOS((p_udiAWOpenAxisErrID = 21570 OR p_udiAWOpenAxisErrID = 21571)
	IF EDGEPOS((p_bAWOpenFwdLmtSen OR p_bAWOpenRevLmtSen OR p_udiAWOpenAxisErrID = 21570 OR p_udiAWOpenAxisErrID = 21571)
		AND tyP0934AW.tyMotionStd.tyBtnJogOpen.bValue = FALSE
		AND tyP0934AW.tyMotionStd.tyBtnJogClose.bValue = FALSE)
	THEN
		fbLmtRstTm.IN	:= TRUE;
	END_IF

	IF fbLmtRstTm.Q = TRUE THEN
		tyP0934AW.tyMotionStd.tyBtnRst.bRtCompl		:= TRUE;
	END_IF

	IF (tyP0934AW.tyMotionStd.tyBtnJogOpen.bValue = FALSE AND tyP0934AW.tyMotionStd.tyBtnJogClose.bValue = FALSE) AND (p_bAWOpenJogging = TRUE) THEN
		bJogStopAW	:= TRUE;
	END_IF

	IF tyP0934AW.tyMotionStd.tyBtnStop.bRtCompl = TRUE THEN
		eAWOpenAct		:= AWActStop;

		IF p_eAWOpenStat = AWActStop AND p_eAWOpenStatus = Done THEN
			eAWOpenAct	:= AWActIdle;

			tyP0934AW.tyMotionStd.tyBtnStop.bRtCompl			:= FALSE;
			tyP0934AW.tyMotionStd.tyBtnJogOpen.bRtCompl			:= FALSE;
			tyP0934AW.tyMotionStd.tyBtnJogClose.bRtCompl		:= FALSE;
			tyP0934AW.tyMotionStd.tyBtnOrigin.bRtCompl			:= FALSE;
			tyP0934AW.tyMotionStd.tyBtnMovAbs.bRtCompl			:= FALSE;
			tyP0934AW.tyMotionStd.tyBtnMovRel.bRtCompl			:= FALSE;
			tyP0934AW.tyAW.tyBtnGo.bRtCompl						:= FALSE;

			tyP0934AW.tyMotionStd.tyBtnStop.bValue				:= TRUE;
			tyP0934AW.tyMotionStd.tyBtnJogOpen.bValue			:= FALSE;
			tyP0934AW.tyMotionStd.tyBtnJogClose.bValue			:= FALSE;
			tyP0934AW.tyMotionStd.tyBtnOrigin.bValue			:= FALSE;
			tyP0934AW.tyMotionStd.tyBtnMovAbs.bValue			:= FALSE;
			tyP0934AW.tyMotionStd.tyBtnMovRel.bValue			:= FALSE;
			tyP0934AW.tyAW.tyBtnGo.bValue						:= FALSE;

			tyP0934AW.tyMotionStd.tyBtnStop.bRtLk				:= TRUE;
			tyP0934AW.tyMotionStd.tyBtnJogOpen.bRtLk			:= FALSE;
			tyP0934AW.tyMotionStd.tyBtnJogClose.bRtLk			:= FALSE;
			tyP0934AW.tyMotionStd.tyBtnOrigin.bRtLk				:= FALSE;
			tyP0934AW.tyMotionStd.tyBtnMovAbs.bRtLk				:= FALSE;
			tyP0934AW.tyMotionStd.tyBtnMovRel.bRtLk				:= FALSE;
			tyP0934AW.tyAW.tyBtnGo.bRtLk						:= FALSE;
		END_IF

	ELSIF (tyP0934AW.tyMotionStd.tyBtnJogOpen.bRtCompl = TRUE) OR (tyP0934AW.tyMotionStd.tyBtnJogClose.bRtCompl = TRUE) OR (bJogStopAW = TRUE) THEN
		bJogSlow					:= FALSE;
		bJogFast					:= FALSE;
		fbJogSlowToFastDlyTm.IN		:= FALSE;

		eAWOpenAct		:= AWActJogStop;

		IF p_eAWOpenStat = AWActJogStop AND p_eAWOpenStatus = Done THEN
			eAWOpenAct	:= AWActIdle;

			bJogStopAW	:= FALSE;

			tyP0934AW.tyMotionStd.tyBtnStop.bRtCompl		:= FALSE;
			tyP0934AW.tyMotionStd.tyBtnJogOpen.bRtCompl		:= FALSE;
			tyP0934AW.tyMotionStd.tyBtnJogClose.bRtCompl	:= FALSE;
			tyP0934AW.tyMotionStd.tyBtnOrigin.bRtCompl		:= FALSE;
			tyP0934AW.tyMotionStd.tyBtnMovAbs.bRtCompl		:= FALSE;
			tyP0934AW.tyMotionStd.tyBtnMovRel.bRtCompl		:= FALSE;
			tyP0934AW.tyAW.tyBtnGo.bRtCompl					:= FALSE;

			tyP0934AW.tyMotionStd.tyBtnStop.bValue			:= TRUE;
			tyP0934AW.tyMotionStd.tyBtnJogOpen.bValue		:= FALSE;
			tyP0934AW.tyMotionStd.tyBtnJogClose.bValue		:= FALSE;
			tyP0934AW.tyMotionStd.tyBtnOrigin.bValue		:= FALSE;
			tyP0934AW.tyMotionStd.tyBtnMovAbs.bValue		:= FALSE;
			tyP0934AW.tyMotionStd.tyBtnMovRel.bValue		:= FALSE;
			tyP0934AW.tyAW.tyBtnGo.bValue					:= FALSE;

			tyP0934AW.tyMotionStd.tyBtnStop.bRtLk			:= TRUE;
			tyP0934AW.tyMotionStd.tyBtnJogOpen.bRtLk		:= FALSE;
			tyP0934AW.tyMotionStd.tyBtnJogClose.bRtLk		:= FALSE;
			tyP0934AW.tyMotionStd.tyBtnOrigin.bRtLk			:= FALSE;
			tyP0934AW.tyMotionStd.tyBtnMovAbs.bRtLk			:= FALSE;
			tyP0934AW.tyMotionStd.tyBtnMovRel.bRtLk			:= FALSE;
			tyP0934AW.tyAW.tyBtnGo.bRtLk					:= FALSE;
		END_IF

	ELSIF tyP0934AW.tyMotionStd.tyBtnPwr.bRtCompl = TRUE THEN
		tyP0934AW.tyMotionStd.tyBtnPwr.bRtLk					:= TRUE;

		IF tyP0934AW.tyMotionStd.tyBtnPwr.bValue = TRUE THEN
			eAWOpenAct		:= AWActPwrOn;

			IF p_eAWOpenStat = AWActPwrOn AND p_eAWOpenStatus = Done THEN
				eAWOpenAct	:= AWActIdle;

				tyP0934AW.tyMotionStd.tyBtnPwr.bRtCompl			:= FALSE;
				tyP0934AW.tyMotionStd.tyBtnPwr.bRtLk			:= FALSE;
			END_IF
		ELSE
			eAWOpenAct		:= AWActPwrOff;

			IF p_eAWOpenStat = AWActPwrOff AND p_eAWOpenStatus = Done THEN
				eAWOpenAct	:= AWActIdle;

				tyP0934AW.tyMotionStd.tyBtnPwr.bRtCompl			:= FALSE;
				tyP0934AW.tyMotionStd.tyBtnPwr.bRtLk			:= FALSE;
			END_IF
		END_IF

	ELSIF tyP0934AW.tyMotionStd.tyBtnOrigin.bRtCompl = TRUE THEN
		tyP0934AW.tyMotionStd.tyBtnOrigin.bValue				:= TRUE;
		tyP0934AW.tyMotionStd.tyBtnStop.bValue					:= FALSE;

		tyP0934AW.tyMotionStd.tyBtnOrigin.bRtLk					:= TRUE;
		tyP0934AW.tyMotionStd.tyBtnStop.bRtLk					:= FALSE;

		eAWOpenAct		:= AWActHoming;

		IF p_eAWOpenStat = AWActHoming AND p_eAWOpenStatus = Done THEN
			eAWOpenAct	:= AWActIdle;

			tyP0934AW.tyMotionStd.tyBtnOrigin.bRtCompl			:= FALSE;
			tyP0934AW.tyMotionStd.tyBtnOrigin.bValue			:= FALSE;
			tyP0934AW.tyMotionStd.tyBtnStop.bValue				:= TRUE;

			tyP0934AW.tyMotionStd.tyBtnOrigin.bRtLk				:= FALSE;
			tyP0934AW.tyMotionStd.tyBtnStop.bRtLk				:= TRUE;
		END_IF

	ELSIF tyP0934AW.tyMotionStd.tyBtnRst.bRtCompl = TRUE THEN
		tyP0934AW.tyMotionStd.tyBtnRst.bValue					:= TRUE;
		tyP0934AW.tyMotionStd.tyBtnRst.bRtLk					:= TRUE;

		eAWOpenAct		:= AWActRstAxisErr;

		IF p_eAWOpenStat = AWActRstAxisErr AND p_eAWOpenStatus = Done THEN
			eAWOpenAct	:= AWActIdle;

			tyP0934AW.tyMotionStd.tyBtnRst.bRtCompl				:= FALSE;
			tyP0934AW.tyMotionStd.tyBtnRst.bValue				:= FALSE;
			tyP0934AW.tyMotionStd.tyBtnRst.bRtLk				:= FALSE;

			fbLmtRstTm.IN			:= FALSE;
		END_IF

	ELSIF tyP0934AW.tyAW.tyBtnGo.bRtCompl = TRUE THEN
		tyP0934AW.tyAW.tyBtnGo.bValue							:= TRUE;
		tyP0934AW.tyMotionStd.tyBtnStop.bValue					:= FALSE;

		tyP0934AW.tyAW.tyBtnGo.bRtLk							:= TRUE;
		tyP0934AW.tyMotionStd.tyBtnStop.bRtLk					:= FALSE;

		diMnlAWGoWidth		:= tyP0934AW.tyAW.tyNumNewWidth.diValue;
		diMnlAWNomSpd		:= tyP0934AW.tyMotionStd.tyNumNomSpd.diValue;

		eAWOpenAct		:= AWActGoWidth;

		IF p_eAWOpenStat = AWActGoWidth AND p_eAWOpenStatus = Done THEN
			eAWOpenAct	:= AWActIdle;

			tyP0934AW.tyAW.tyBtnGo.bRtCompl						:= FALSE;
			tyP0934AW.tyAW.tyBtnGo.bValue						:= FALSE;
			tyP0934AW.tyMotionStd.tyBtnStop.bValue				:= TRUE;

			tyP0934AW.tyAW.tyBtnGo.bRtLk						:= FALSE;
			tyP0934AW.tyMotionStd.tyBtnStop.bRtLk				:= TRUE;
		END_IF

	ELSIF tyP0934AW.tyMotionStd.tyBtnMovAbs.bRtCompl = TRUE THEN
		tyP0934AW.tyMotionStd.tyBtnMovAbs.bValue				:= TRUE;
		tyP0934AW.tyMotionStd.tyBtnStop.bValue					:= FALSE;

		tyP0934AW.tyMotionStd.tyBtnMovAbs.bRtLk					:= TRUE;
		tyP0934AW.tyMotionStd.tyBtnStop.bRtLk					:= FALSE;

		diMnlAWTargetPos	:= tyP0934AW.tyMotionStd.tyNumTargetPos.diValue;
		diMnlAWNomSpd		:= tyP0934AW.tyMotionStd.tyNumNomSpd.diValue;

		eAWOpenAct		:= AWActMovAbs;

		IF p_eAWOpenStat = AWActMovAbs AND p_eAWOpenStatus = Done THEN
			eAWOpenAct	:= AWActIdle;

			tyP0934AW.tyMotionStd.tyBtnMovAbs.bRtCompl			:= FALSE;
			tyP0934AW.tyMotionStd.tyBtnMovAbs.bValue			:= FALSE;
			tyP0934AW.tyMotionStd.tyBtnStop.bValue				:= TRUE;

			tyP0934AW.tyMotionStd.tyBtnMovAbs.bRtLk				:= FALSE;
			tyP0934AW.tyMotionStd.tyBtnStop.bRtLk				:= TRUE;
		END_IF

	ELSIF tyP0934AW.tyMotionStd.tyBtnMovRel.bRtCompl = TRUE THEN
		tyP0934AW.tyMotionStd.tyBtnMovRel.bValue				:= TRUE;
		tyP0934AW.tyMotionStd.tyBtnStop.bValue					:= FALSE;

		tyP0934AW.tyMotionStd.tyBtnMovRel.bRtLk					:= TRUE;
		tyP0934AW.tyMotionStd.tyBtnStop.bRtLk					:= FALSE;

		diMnlAWStepSize		:= tyP0934AW.tyMotionStd.tyNumStepSize.diValue;
		diMnlAWNomSpd		:= tyP0934AW.tyMotionStd.tyNumNomSpd.diValue;

		eAWOpenAct		:= AWActMovRel;

		IF p_eAWOpenStat = AWActMovRel AND p_eAWOpenStatus = Done THEN
			eAWOpenAct	:= AWActIdle;

			tyP0934AW.tyMotionStd.tyBtnMovRel.bRtCompl			:= FALSE;
			tyP0934AW.tyMotionStd.tyBtnMovRel.bValue			:= FALSE;
			tyP0934AW.tyMotionStd.tyBtnStop.bValue				:= TRUE;

			tyP0934AW.tyMotionStd.tyBtnMovRel.bRtLk				:= FALSE;
			tyP0934AW.tyMotionStd.tyBtnStop.bRtLk				:= TRUE;
		END_IF

	ELSIF (tyP0934AW.tyMotionStd.tyBtnJogOpen.bValue = TRUE) AND (fbJogSlowToFastDlyTm.Q = FALSE) AND (bJogSlow = FALSE) THEN
		tyP0934AW.tyMotionStd.tyBtnStop.bValue					:= FALSE;
		tyP0934AW.tyMotionStd.tyBtnStop.bRtLk					:= FALSE;

		fbJogSlowToFastDlyTm.IN		:= TRUE;

		diMnlAWJogSpd		:= tyP0934AW.tyMotionStd.tyNumSlwSpd.diValue;

		eAWOpenAct		:= AWActJogOpen;

		IF p_eAWOpenStat = AWActJogOpen AND p_eAWOpenStatus = Done THEN
			eAWOpenAct	:= AWActIdle;
			bJogSlow				:= TRUE;
		ELSIF p_eAWOpenStatus = Error THEN
			fbJogSlowToFastDlyTm.IN	:= FALSE;
			bJogSlow				:= TRUE;
		END_IF

	ELSIF (tyP0934AW.tyMotionStd.tyBtnJogOpen.bValue = TRUE) AND (fbJogSlowToFastDlyTm.Q = TRUE) AND (bJogFast = FALSE) THEN
		tyP0934AW.tyMotionStd.tyBtnStop.bValue					:= FALSE;
		tyP0934AW.tyMotionStd.tyBtnStop.bRtLk					:= FALSE;

		fbJogSlowToFastDlyTm.IN		:= TRUE;

		diMnlAWJogSpd		:= tyP0934AW.tyMotionStd.tyNumNomSpd.diValue;

		eAWOpenAct		:= AWActJogOpen;

		IF p_eAWOpenStat = AWActJogOpen AND p_eAWOpenStatus = Done THEN
			eAWOpenAct	:= AWActIdle;
			bJogFast				:= TRUE;
		ELSIF p_eAWOpenStatus = Error THEN
			fbJogSlowToFastDlyTm.IN	:= FALSE;
			bJogFast				:= TRUE;
		END_IF

	ELSIF (tyP0934AW.tyMotionStd.tyBtnJogClose.bValue = TRUE) AND (fbJogSlowToFastDlyTm.Q = FALSE) AND (bJogSlow = FALSE) THEN
		tyP0934AW.tyMotionStd.tyBtnStop.bValue					:= FALSE;
		tyP0934AW.tyMotionStd.tyBtnStop.bRtLk					:= FALSE;

		fbJogSlowToFastDlyTm.IN		:= TRUE;

		diMnlAWJogSpd		:= tyP0934AW.tyMotionStd.tyNumSlwSpd.diValue;

		eAWOpenAct		:= AWActJogClose;

		IF p_eAWOpenStat = AWActJogClose AND p_eAWOpenStatus = Done THEN
			eAWOpenAct	:= AWActIdle;
			bJogSlow				:= TRUE;
		ELSIF p_eAWOpenStatus = Error THEN
			fbJogSlowToFastDlyTm.IN	:= FALSE;
			bJogSlow				:= TRUE;
		END_IF

	ELSIF (tyP0934AW.tyMotionStd.tyBtnJogClose.bValue = TRUE) AND (fbJogSlowToFastDlyTm.Q = TRUE) AND (bJogFast = FALSE) THEN
		tyP0934AW.tyMotionStd.tyBtnStop.bValue					:= FALSE;
		tyP0934AW.tyMotionStd.tyBtnStop.bRtLk					:= FALSE;

		fbJogSlowToFastDlyTm.IN		:= TRUE;

		diMnlAWJogSpd		:= tyP0934AW.tyMotionStd.tyNumNomSpd.diValue;

		eAWOpenAct		:= AWActJogClose;

		IF p_eAWOpenStat = AWActJogClose AND p_eAWOpenStatus = Done THEN
			eAWOpenAct	:= AWActIdle;
			bJogFast				:= TRUE;
		ELSIF p_eAWOpenStatus = Error THEN
			fbJogSlowToFastDlyTm.IN	:= FALSE;
			bJogFast				:= TRUE;
		END_IF
	END_IF

	//Shutter Control
	IF tyP0934AW.tyInOutletShutterFB.tyBtnOpen.bRtCompl = TRUE THEN
		tyP0934AW.tyInOutletShutterFB.tyBtnOpen.bRtCompl	:= FALSE;

		tyP0934AW.tyInOutletShutterFB.tyBtnOpen.bValue	:= TRUE;
		tyP0934AW.tyInOutletShutterFB.tyBtnClose.bValue	:= FALSE;

	ELSIF tyP0934AW.tyInOutletShutterFB.tyBtnClose.bRtCompl = TRUE THEN
		tyP0934AW.tyInOutletShutterFB.tyBtnClose.bRtCompl	:= FALSE;

		tyP0934AW.tyInOutletShutterFB.tyBtnClose.bValue	:= TRUE;
		tyP0934AW.tyInOutletShutterFB.tyBtnOpen.bValue	:= FALSE;
	END_IF

	IF tyP0934AW.tyInOutletShutterFB.tyBtnOpen.bValue = TRUE THEN
		eInShutterAct	:= PneuActRet;
		eOutShutterAct	:= PneuActRet;

		IF (p_eInShutterStat = PneuActRet AND p_eInShutterStatus = Done)
			AND (p_eOutShutterStat = PneuActRet AND p_eOutShutterStatus = Done)
			THEN
			eInShutterAct	:= PneuActIdle;
			eOutShutterAct	:= PneuActIdle;
			tyP0934AW.tyInOutletShutterFB.tyBtnOpen.bValue	:= FALSE;
		ELSIF p_eInShutterStatus = Error OR p_eOutShutterStatus = Error THEN
			tyP0934AW.tyInOutletShutterFB.tyBtnOpen.bValue	:= FALSE;
		END_IF

	ELSIF tyP0934AW.tyInOutletShutterFB.tyBtnClose.bValue = TRUE THEN
		eInShutterAct	:= PneuActExt;
		eOutShutterAct	:= PneuActExt;
		IF (p_eInShutterStat = PneuActExt AND p_eInShutterStatus = Done)
			AND (p_eOutShutterStat = PneuActExt AND p_eOutShutterStatus = Done)
			THEN
			eInShutterAct	:= PneuActIdle;
			eOutShutterAct	:= PneuActIdle;
			tyP0934AW.tyInOutletShutterFB.tyBtnClose.bValue := FALSE;
		ELSIF p_eInShutterStatus = Error OR p_eOutShutterStatus = Error THEN
			tyP0934AW.tyInOutletShutterFB.tyBtnClose.bValue := FALSE;
		END_IF
	END_IF

END_ACTION
```

#### Act_OptP0934FullMask.st
```iecst
ACTION Act_OptP0934FullMask:

	IF eCurrPage = UIP0934AW THEN

		IF p_tyDI.bEStopSig = FALSE THEN
			p_tyC0002FullMask ACCESS ADR(tyP0934AW.tyFullMaskEStop);

		ELSIF p_tyDI.bCoverSWSig = FALSE THEN
			p_tyC0002FullMask ACCESS ADR(tyP0934AW.tyFullMaskCWSig);

		ELSIF p_tyDI.bSafetyRlySig = FALSE THEN
			p_tyC0002FullMask ACCESS ADR(tyP0934AW.tyFullMaskSafetyRly);

		ELSIF p_tyDI.bConvLftSen THEN
			p_tyC0002FullMask ACCESS ADR(tyP0934AW.tyFullMaskLftSenInterrupt);

		ELSIF p_tyDI.bConvRgtSen THEN
			p_tyC0002FullMask ACCESS ADR(tyP0934AW.tyFullMaskRgtSenInterrupt);

		ELSIF p_tyNtParamCurr.bProjInletShutPrep AND (p_tyDI.bInShutterCloseRS = FALSE
			OR (p_tyDI.bInShutterCloseRS2 = FALSE AND p_tyNtParamCurr.tyDISettings.diInShutterCloseRS2 > 0)
			OR (p_tyDI.bInShutterCloseRS3 = FALSE AND p_tyNtParamCurr.tyDISettings.diInShutterCloseRS3 > 0)) THEN
			IF p_tyNtParamCurr.bProjCurtainSenPrep THEN
				IF p_tyDI.bInShutterCloseRS = FALSE OR p_tyDI.bInShutterCloseRS2 = FALSE OR p_tyDI.bInShutterCloseRS3 = FALSE THEN
					p_tyC0002FullMask ACCESS ADR(tyP0934AW.tyFullMaskInShutOpnInterrupt);
				END_IF
			ELSE
				IF p_tyDI.bInShutterCloseRS = FALSE THEN
					p_tyC0002FullMask ACCESS ADR(tyP0934AW.tyFullMaskInShutOpnInterrupt);
				END_IF
			END_IF

	//	ELSIF p_tyNtParamCurr.bProjOutletShutPrep AND p_tyDI.bOutShutterCloseRS = FALSE AND p_McParamOutShutterDis = FALSE THEN
		ELSIF p_tyNtParamCurr.bProjOutletShutPrep AND p_tyDI.bOutShutterCloseRS = FALSE  THEN
			p_tyC0002FullMask ACCESS ADR(tyP0934AW.tyFullMaskOutShutOpnInterrupt);

		ELSIF  p_tyDI.bPullerRetRS = FALSE THEN
			p_tyC0002FullMask ACCESS ADR(tyP0934AW.tyFullMaskPullerRetInterrupt);

		ELSE
			p_tyC0002FullMask ACCESS ADR(tyP0934AW.tyFullMaskHide);

		END_IF

	END_IF

END_ACTION
```
